LIN {X 0,Y 220.837,Z 392.973,A -85,B 0,C 180,E1 -20401.487,E2 -20401.487} C_VEL
LIN {X 0,Y 220.874,Z 392.97,A -85,B 0,C 180,E1 -20405.566,E2 -20405.566} C_VEL
LIN {X 0,Y 220.912,Z 392.963,A -85,B 0,C 180,E1 -20409.516,E2 -20409.516} C_VEL
LIN {X 0,Y 221.019,Z 392.952,A -85,B 0,C 180,E1 -20413.371,E2 -20413.371} C_VEL
LIN {X 0,Y 221.114,Z 392.939,A -85,B 0,C 180,E1 -20419.006,E2 -20419.006} C_VEL
LIN {X 0,Y 221.291,Z 392.918,A -85,B 0,C 180,E1 -20422.702,E2 -20422.702} C_VEL
LIN {X 0,Y 221.515,Z 392.893,A -85,B 0,C 180,E1 -20428.182,E2 -20428.182} C_VEL
LIN {X 0,Y 221.515,Z 392.893,A -85,B 0,C 180,E1 -20431.818,E2 -20431.818} C_VEL
LIN {X 0,Y 221.262,Z 392.922,A -85,B 0,C 180,E1 -20437.3,E2 -20437.3} C_VEL
LIN {X 0,Y 221.084,Z 392.943,A -85,B 0,C 180,E1 -20440.996,E2 -20440.996} C_VEL
LIN {X 0,Y 221.019,Z 392.952,A -85,B 0,C 180,E1 -20446.63,E2 -20446.63} C_VEL
LIN {X 0,Y 220.896,Z 392.965,A -85,B 0,C 180,E1 -20450.486,E2 -20450.486} C_VEL
LIN {X 0,Y 220.87,Z 392.97,A -85,B 0,C 180,E1 -20454.435,E2 -20454.435} C_VEL
LIN {X 0,Y 220.838,Z 392.973,A -85,B 0,C 180,E1 -20458.514,E2 -20458.514} C_VEL
LIN {X 0,Y 220.827,Z 392.976,A -85,B 0,C 180,E1 -20462.755,E2 -20462.755} C_VEL
LIN {X 0,Y 220.841,Z 392.976,A -85,B 0,C 180,E1 -20467.288,E2 -20467.288} C_VEL
LIN {X 0,Y 220.778,Z 392.982,A -85,B 0,C 180,E1 -20471.951,E2 -20471.951} C_VEL
LIN {X 0,Y 220.778,Z 392.982,A -85,B 0,C 180,E1 -20475.547,E2 -20475.547} C_VEL
LIN {X 0,Y 220.809,Z 392.978,A -85,B 0,C 180,E1 -20480.463,E2 -20480.463} C_VEL
LIN {X 0,Y 220.897,Z 392.967,A -85,B 0,C 180,E1 -20485.062,E2 -20485.062} C_VEL
LIN {X 0,Y 221.191,Z 393.123,A -85,B 0,C 180,E1 -20488.024,E2 -20488.024} C_VEL
LIN {X 0,Y 221.094,Z 396.042,A -85,B 0,C 180,E1 -20490.481,E2 -20490.481} C_VEL
LIN {X 0,Y 220.516,Z 400.977,A -85,B 0,C 180,E1 -20494.516,E2 -20494.516} C_VEL
LIN {X 0,Y 219.978,Z 407.083,A -85,B 0,C 180,E1 -20499.425,E2 -20499.425} C_VEL
LIN {X 0,Y 219.573,Z 412.628,A -85,B 0,C 180,E1 -20503.788,E2 -20503.788} C_VEL
LIN {X 0,Y 219.439,Z 417.082,A -85,B 0,C 180,E1 -20507.162,E2 -20507.162} C_VEL
LIN {X 0,Y 220.425,Z 428.94,A -85,B 0,C 180,E1 -20508.389,E2 -20508.389} C_VEL
LIN {X 0,Y 221.015,Z 435.556,A -85,B 0,C 180,E1 -20509.233,E2 -20509.233} C_VEL
LIN {X 0,Y 220.496,Z 447.027,A -85,B 0,C 180,E1 -20511.038,E2 -20511.038} C_VEL
LIN {X 0,Y 220.001,Z 457.347,A -85,B 0,C 180,E1 -20513.12,E2 -20513.12} C_VEL
LIN {X 0,Y 219.741,Z 464.712,A -85,B 0,C 180,E1 -20514.954,E2 -20514.954} C_VEL
LIN {X 0,Y 219.303,Z 472.284,A -85,B 0,C 180,E1 -20517.245,E2 -20517.245} C_VEL
LIN {X 0,Y 219.233,Z 478.476,A -85,B 0,C 180,E1 -20519.541,E2 -20519.541} C_VEL
LIN {X 0,Y 219.511,Z 483.38,A -85,B 0,C 180,E1 -20521.835,E2 -20521.835} C_VEL
LIN {X 0,Y 220.284,Z 487.936,A -85,B 0,C 180,E1 -20524.575,E2 -20524.575} C_VEL
LIN {X 0,Y 221.64,Z 491.134,A -85,B 0,C 180,E1 -20527.287,E2 -20527.287} C_VEL
LIN {X 0,Y 222.837,Z 492.539,A -85,B 0,C 180,E1 -20529.073,E2 -20529.073} C_VEL
LIN {X 0,Y 224.278,Z 493.429,A -85,B 0,C 180,E1 -20530.837,E2 -20530.837} C_VEL
LIN {X 0,Y 226.104,Z 493.732,A -85,B 0,C 180,E1 -20532.567,E2 -20532.567} C_VEL
LIN {X 0,Y 228.077,Z 493.509,A -85,B 0,C 180,E1 -20534.271,E2 -20534.271} C_VEL
LIN {X 0,Y 230.273,Z 492.801,A -85,B 0,C 180,E1 -20535.943,E2 -20535.943} C_VEL
LIN {X 0,Y 232.689,Z 491.534,A -85,B 0,C 180,E1 -20537.58,E2 -20537.58} C_VEL
LIN {X 0,Y 236.667,Z 488.649,A -85,B 0,C 180,E1 -20539.968,E2 -20539.968} C_VEL
LIN {X 0,Y 241.113,Z 484.562,A -85,B 0,C 180,E1 -20542.267,E2 -20542.267} C_VEL
LIN {X 0,Y 244.319,Z 481.041,A -85,B 0,C 180,E1 -20543.748,E2 -20543.748} C_VEL
LIN {X 0,Y 246.024,Z 477.848,A -85,B 0,C 180,E1 -20545.372,E2 -20545.372} C_VEL
LIN {X 0,Y 247.77,Z 472.241,A -85,B 0,C 180,E1 -20548.439,E2 -20548.439} C_VEL
LIN {X 0,Y 248.776,Z 467.147,A -85,B 0,C 180,E1 -20551.482,E2 -20551.482} C_VEL
LIN {X 0,Y 249.086,Z 464.573,A -85,B 0,C 180,E1 -20553.264,E2 -20553.264} C_VEL
LIN {X 0,Y 249.164,Z 462.654,A -85,B 0,C 180,E1 -20555.116,E2 -20555.116} C_VEL
LIN {X 0,Y 249.105,Z 460.856,A -85,B 0,C 180,E1 -20557.817,E2 -20557.817} C_VEL
LIN {X 0,Y 249.25,Z 460.084,A -85,B 0,C 180,E1 -20560.43,E2 -20560.43} C_VEL
LIN {X 0,Y 249.561,Z 460.468,A -85,B 0,C 180,E1 -20562.928,E2 -20562.928} C_VEL
LIN {X 0,Y 249.989,Z 461.962,A -85,B 0,C 180,E1 -20565.345,E2 -20565.345} C_VEL
LIN {X 0,Y 251.219,Z 465.936,A -85,B 0,C 180,E1 -20569.055,E2 -20569.055} C_VEL
LIN {X 0,Y 251.946,Z 468.627,A -85,B 0,C 180,E1 -20570.815,E2 -20570.815} C_VEL
LIN {X 0,Y 252.423,Z 471.374,A -85,B 0,C 180,E1 -20572.227,E2 -20572.227} C_VEL
LIN {X 0,Y 250.398,Z 479.099,A -85,B 0,C 180,E1 -20574.484,E2 -20574.484} C_VEL
LIN {X 0,Y 247.406,Z 487.692,A -85,B 0,C 180,E1 -20576.883,E2 -20576.883} C_VEL
LIN {X 0,Y 244.808,Z 493.219,A -85,B 0,C 180,E1 -20578.404,E2 -20578.404} C_VEL
LIN {X 0,Y 239.832,Z 501.02,A -85,B 0,C 180,E1 -20580.604,E2 -20580.604} C_VEL
LIN {X 0,Y 234.051,Z 508.808,A -85,B 0,C 180,E1 -20583.353,E2 -20583.353} C_VEL
LIN {X 0,Y 231.481,Z 511.607,A -85,B 0,C 180,E1 -20584.482,E2 -20584.482} C_VEL
LIN {X 0,Y 225.685,Z 515.698,A -85,B 0,C 180,E1 -20586.229,E2 -20586.229} C_VEL
LIN {X 0,Y 220.118,Z 519.017,A -85,B 0,C 180,E1 -20588.141,E2 -20588.141} C_VEL
LIN {X 0,Y 217.954,Z 520.611,A -85,B 0,C 180,E1 -20589.505,E2 -20589.505} C_VEL
LIN {X 0,Y 215.082,Z 523.55,A -85,B 0,C 180,E1 -20592.897,E2 -20592.897} C_VEL
LIN {X 0,Y 213.022,Z 525.29,A -85,B 0,C 180,E1 -20596.647,E2 -20596.647} C_VEL
LIN {X 0,Y 212.308,Z 525.696,A -85,B 0,C 180,E1 -20600.472,E2 -20600.472} C_VEL
LIN {X 0,Y 212.513,Z 524.63,A -85,B 0,C 180,E1 -20604.306,E2 -20604.306} C_VEL
LIN {X 0,Y 212.841,Z 523.547,A -85,B 0,C 180,E1 -20606.213,E2 -20606.213} C_VEL
LIN {X 0,Y 213.518,Z 521.058,A -85,B 0,C 180,E1 -20609.057,E2 -20609.057} C_VEL
LIN {X 0,Y 213.859,Z 517.355,A -85,B 0,C 180,E1 -20611.883,E2 -20611.883} C_VEL
LIN {X 0,Y 213.773,Z 512.137,A -85,B 0,C 180,E1 -20614.714,E2 -20614.714} C_VEL
LIN {X 0,Y 213.693,Z 506.567,A -85,B 0,C 180,E1 -20617.084,E2 -20617.084} C_VEL
LIN {X 0,Y 213.821,Z 498.336,A -85,B 0,C 180,E1 -20619.888,E2 -20619.888} C_VEL
LIN {X 0,Y 214.203,Z 488.282,A -85,B 0,C 180,E1 -20622.554,E2 -20622.554} C_VEL
LIN {X 0,Y 214.869,Z 478.168,A -85,B 0,C 180,E1 -20624.684,E2 -20624.684} C_VEL
LIN {X 0,Y 215.276,Z 471.414,A -85,B 0,C 180,E1 -20625.867,E2 -20625.867} C_VEL
LIN {X 0,Y 214.305,Z 459.661,A -85,B 0,C 180,E1 -20627.479,E2 -20627.479} C_VEL
LIN {X 0,Y 213.616,Z 447.834,A -85,B 0,C 180,E1 -20628.736,E2 -20628.736} C_VEL
LIN {X 0,Y 213.55,Z 435.845,A -85,B 0,C 180,E1 -20629.714,E2 -20629.714} C_VEL
LIN {X 0,Y 215.596,Z 424.642,A -85,B 0,C 180,E1 -20636.108,E2 -20636.108} C_VEL
LIN {X 0,Y 217.998,Z 415.833,A -85,B 0,C 180,E1 -20641.052,E2 -20641.052} C_VEL
LIN {X 0,Y 218.142,Z 414.232,A -85,B 0,C 180,E1 -20641.952,E2 -20641.952} C_VEL
LIN {X 0,Y 216.248,Z 405.804,A -85,B 0,C 180,E1 -20646.958,E2 -20646.958} C_VEL
LIN {X 0,Y 214.577,Z 397.868,A -85,B 0,C 180,E1 -20651.831,E2 -20651.831} C_VEL
LIN {X 0,Y 213.832,Z 393.846,A -85,B 0,C 180,E1 -20654.536,E2 -20654.536} C_VEL
LIN {X 0,Y 213.723,Z 393.86,A -85,B 0,C 180,E1 -20659.141,E2 -20659.141} C_VEL
LIN {X 0,Y 213.753,Z 393.858,A -85,B 0,C 180,E1 -20663.713,E2 -20663.713} C_VEL
LIN {X 0,Y 213.77,Z 393.857,A -85,B 0,C 180,E1 -20668.263,E2 -20668.263} C_VEL
LIN {X 0,Y 213.826,Z 393.847,A -85,B 0,C 180,E1 -20672.603,E2 -20672.603} C_VEL
LIN {X 0,Y 213.852,Z 393.844,A -85,B 0,C 180,E1 -20676.953,E2 -20676.953} C_VEL
LIN {X 0,Y 213.944,Z 393.829,A -85,B 0,C 180,E1 -20682.804,E2 -20682.804} C_VEL
LIN {X 0,Y 213.981,Z 393.829,A -85,B 0,C 180,E1 -20686.708,E2 -20686.708} C_VEL
LIN {X 0,Y 214.197,Z 393.799,A -85,B 0,C 180,E1 -20690.558,E2 -20690.558} C_VEL
LIN {X 0,Y 214.249,Z 393.793,A -85,B 0,C 180,E1 -20692.46,E2 -20692.46} C_VEL
LIN {X 0,Y 214.449,Z 393.769,A -85,B 0,C 180,E1 -20698.122,E2 -20698.122} C_VEL
LIN {X 0,Y 214.552,Z 393.756,A -85,B 0,C 180,E1 -20700,E2 -20700} C_VEL
LIN {X 0,Y 214.447,Z 393.771,A -85,B 0,C 180,E1 -20701.878,E2 -20701.878} C_VEL
LIN {X 0,Y 214.249,Z 393.794,A -85,B 0,C 180,E1 -20707.54,E2 -20707.54} C_VEL
LIN {X 0,Y 214.048,Z 393.823,A -85,B 0,C 180,E1 -20711.362,E2 -20711.362} C_VEL
LIN {X 0,Y 213.935,Z 393.836,A -85,B 0,C 180,E1 -20715.237,E2 -20715.237} C_VEL
LIN {X 0,Y 213.869,Z 393.844,A -85,B 0,C 180,E1 -20719.185,E2 -20719.185} C_VEL
LIN {X 0,Y 213.848,Z 393.847,A -85,B 0,C 180,E1 -20723.227,E2 -20723.227} C_VEL
LIN {X 0,Y 213.829,Z 393.848,A -85,B 0,C 180,E1 -20727.45,E2 -20727.45} C_VEL
LIN {X 0,Y 213.777,Z 393.854,A -85,B 0,C 180,E1 -20731.736,E2 -20731.736} C_VEL
LIN {X 0,Y 213.744,Z 393.857,A -85,B 0,C 180,E1 -20736.288,E2 -20736.288} C_VEL
LIN {X 0,Y 213.713,Z 393.862,A -85,B 0,C 180,E1 -20741.125,E2 -20741.125} C_VEL
LIN {X 0,Y 213.708,Z 393.86,A -85,B 0,C 180,E1 -20743.678,E2 -20743.678} C_VEL
LIN {X 0,Y 213.71,Z 393.864,A -85,B 0,C 180,E1 -20746.343,E2 -20746.343} C_VEL
LIN {X 0,Y 213.737,Z 393.856,A -85,B 0,C 180,E1 -20751.336,E2 -20751.336} C_VEL
LIN {X 0,Y 213.771,Z 393.856,A -85,B 0,C 180,E1 -20756.021,E2 -20756.021} C_VEL
LIN {X 0,Y 213.782,Z 393.853,A -85,B 0,C 180,E1 -20760.454,E2 -20760.454} C_VEL
LIN {X 0,Y 213.806,Z 393.852,A -85,B 0,C 180,E1 -20764.703,E2 -20764.703} C_VEL
LIN {X 0,Y 213.843,Z 393.844,A -85,B 0,C 180,E1 -20768.807,E2 -20768.807} C_VEL
LIN {X 0,Y 213.947,Z 393.834,A -85,B 0,C 180,E1 -20772.804,E2 -20772.804} C_VEL
LIN {X 0,Y 213.983,Z 393.826,A -85,B 0,C 180,E1 -20776.709,E2 -20776.709} C_VEL
LIN {X 0,Y 214.169,Z 393.807,A -85,B 0,C 180,E1 -20780.557,E2 -20780.557} C_VEL
LIN {X 0,Y 214.229,Z 393.799,A -85,B 0,C 180,E1 -20782.46,E2 -20782.46} C_VEL
LIN {X 0,Y 214.448,Z 393.773,A -85,B 0,C 180,E1 -20788.122,E2 -20788.122} C_VEL
LIN {X 0,Y 214.557,Z 393.761,A -85,B 0,C 180,E1 -20790,E2 -20790} C_VEL
LIN {X 0,Y 214.448,Z 393.773,A -85,B 0,C 180,E1 -20791.878,E2 -20791.878} C_VEL
LIN {X 0,Y 214.201,Z 393.802,A -85,B 0,C 180,E1 -20797.542,E2 -20797.542} C_VEL
LIN {X 0,Y 214.01,Z 393.825,A -85,B 0,C 180,E1 -20801.364,E2 -20801.364} C_VEL
LIN {X 0,Y 213.937,Z 393.834,A -85,B 0,C 180,E1 -20805.237,E2 -20805.237} C_VEL
LIN {X 0,Y 213.871,Z 393.843,A -85,B 0,C 180,E1 -20809.185,E2 -20809.185} C_VEL
LIN {X 0,Y 213.85,Z 393.844,A -85,B 0,C 180,E1 -20813.227,E2 -20813.227} C_VEL
LIN {X 0,Y 213.831,Z 393.85,A -85,B 0,C 180,E1 -20817.45,E2 -20817.45} C_VEL
LIN {X 0,Y 213.782,Z 393.855,A -85,B 0,C 180,E1 -20821.736,E2 -20821.736} C_VEL
LIN {X 0,Y 213.755,Z 393.856,A -85,B 0,C 180,E1 -20826.287,E2 -20826.287} C_VEL
LIN {X 0,Y 213.72,Z 393.862,A -85,B 0,C 180,E1 -20831.124,E2 -20831.124} C_VEL
LIN {X 0,Y 213.712,Z 393.863,A -85,B 0,C 180,E1 -20833.678,E2 -20833.678} C_VEL
LIN {X 0,Y 213.71,Z 393.86,A -85,B 0,C 180,E1 -20836.344,E2 -20836.344} C_VEL
LIN {X 0,Y 213.737,Z 393.862,A -85,B 0,C 180,E1 -20841.336,E2 -20841.336} C_VEL
LIN {X 0,Y 214.031,Z 393.818,A -85,B 0,C 180,E1 -20847.194,E2 -20847.194} C_VEL
LIN {X 0,Y 214.158,Z 393.995,A -85,B 0,C 180,E1 -20848.05,E2 -20848.05} C_VEL
LIN {X 0,Y 214.035,Z 396.832,A -85,B 0,C 180,E1 -20850.492,E2 -20850.492} C_VEL
LIN {X 0,Y 213.308,Z 403.024,A -85,B 0,C 180,E1 -20855.679,E2 -20855.679} C_VEL
LIN {X 0,Y 212.782,Z 409.154,A -85,B 0,C 180,E1 -20860.713,E2 -20860.713} C_VEL
LIN {X 0,Y 212.369,Z 415.285,A -85,B 0,C 180,E1 -20865.629,E2 -20865.629} C_VEL
LIN {X 0,Y 212.342,Z 417.279,A -85,B 0,C 180,E1 -20867.212,E2 -20867.212} C_VEL
LIN {X 0,Y 213.576,Z 431.068,A -85,B 0,C 180,E1 -20868.733,E2 -20868.733} C_VEL
LIN {X 0,Y 213.93,Z 435.64,A -85,B 0,C 180,E1 -20869.351,E2 -20869.351} C_VEL
LIN {X 0,Y 213.428,Z 446.255,A -85,B 0,C 180,E1 -20871.071,E2 -20871.071} C_VEL
LIN {X 0,Y 212.946,Z 456.398,A -85,B 0,C 180,E1 -20873.129,E2 -20873.129} C_VEL
LIN {X 0,Y 212.615,Z 464.917,A -85,B 0,C 180,E1 -20875.26,E2 -20875.26} C_VEL
LIN {X 0,Y 212.225,Z 472.594,A -85,B 0,C 180,E1 -20877.628,E2 -20877.628} C_VEL
LIN {X 0,Y 212.233,Z 479.859,A -85,B 0,C 180,E1 -20880.474,E2 -20880.474} C_VEL
LIN {X 0,Y 212.64,Z 484.667,A -85,B 0,C 180,E1 -20882.842,E2 -20882.842} C_VEL
LIN {X 0,Y 213.582,Z 489.1,A -85,B 0,C 180,E1 -20885.665,E2 -20885.665} C_VEL
LIN {X 0,Y 214.601,Z 491.312,A -85,B 0,C 180,E1 -20887.527,E2 -20887.527} C_VEL
LIN {X 0,Y 215.856,Z 492.951,A -85,B 0,C 180,E1 -20889.369,E2 -20889.369} C_VEL
LIN {X 0,Y 217.355,Z 494.052,A -85,B 0,C 180,E1 -20891.187,E2 -20891.187} C_VEL
LIN {X 0,Y 219.226,Z 494.623,A -85,B 0,C 180,E1 -20892.968,E2 -20892.968} C_VEL
LIN {X 0,Y 221.303,Z 494.639,A -85,B 0,C 180,E1 -20894.718,E2 -20894.718} C_VEL
LIN {X 0,Y 223.58,Z 494.155,A -85,B 0,C 180,E1 -20896.434,E2 -20896.434} C_VEL
LIN {X 0,Y 226.106,Z 493.159,A -85,B 0,C 180,E1 -20898.109,E2 -20898.109} C_VEL
LIN {X 0,Y 230.231,Z 490.713,A -85,B 0,C 180,E1 -20900.551,E2 -20900.551} C_VEL
LIN {X 0,Y 234.838,Z 487.053,A -85,B 0,C 180,E1 -20902.895,E2 -20902.895} C_VEL
LIN {X 0,Y 238.186,Z 483.92,A -85,B 0,C 180,E1 -20904.399,E2 -20904.399} C_VEL
LIN {X 0,Y 239.438,Z 482.364,A -85,B 0,C 180,E1 -20905.189,E2 -20905.189} C_VEL
LIN {X 0,Y 241.512,Z 478.123,A -85,B 0,C 180,E1 -20907.749,E2 -20907.749} C_VEL
LIN {X 0,Y 243.002,Z 473.908,A -85,B 0,C 180,E1 -20910.405,E2 -20910.405} C_VEL
LIN {X 0,Y 244.081,Z 470.048,A -85,B 0,C 180,E1 -20913.167,E2 -20913.167} C_VEL
LIN {X 0,Y 244.456,Z 468.089,A -85,B 0,C 180,E1 -20915.099,E2 -20915.099} C_VEL
LIN {X 0,Y 244.601,Z 466.776,A -85,B 0,C 180,E1 -20917.113,E2 -20917.113} C_VEL
LIN {X 0,Y 244.753,Z 465.998,A -85,B 0,C 180,E1 -20919.177,E2 -20919.177} C_VEL
LIN {X 0,Y 245.103,Z 465.903,A -85,B 0,C 180,E1 -20921.796,E2 -20921.796} C_VEL
LIN {X 0,Y 245.476,Z 466.939,A -85,B 0,C 180,E1 -20924.294,E2 -20924.294} C_VEL
LIN {X 0,Y 245.926,Z 468.963,A -85,B 0,C 180,E1 -20926.696,E2 -20926.696} C_VEL
LIN {X 0,Y 246.716,Z 471.544,A -85,B 0,C 180,E1 -20929.066,E2 -20929.066} C_VEL
LIN {X 0,Y 247.32,Z 475.087,A -85,B 0,C 180,E1 -20931.305,E2 -20931.305} C_VEL
LIN {X 0,Y 247.341,Z 475.694,A -85,B 0,C 180,E1 -20931.619,E2 -20931.619} C_VEL
LIN {X 0,Y 245.205,Z 482.097,A -85,B 0,C 180,E1 -20933.613,E2 -20933.613} C_VEL
LIN {X 0,Y 241.251,Z 491.306,A -85,B 0,C 180,E1 -20936.392,E2 -20936.392} C_VEL
LIN {X 0,Y 237.333,Z 497.714,A -85,B 0,C 180,E1 -20938.29,E2 -20938.29} C_VEL
LIN {X 0,Y 231.235,Z 505.657,A -85,B 0,C 180,E1 -20940.902,E2 -20940.902} C_VEL
LIN {X 0,Y 226.595,Z 511.194,A -85,B 0,C 180,E1 -20943.273,E2 -20943.273} C_VEL
LIN {X 0,Y 221.355,Z 517.034,A -85,B 0,C 180,E1 -20946.617,E2 -20946.617} C_VEL
LIN {X 0,Y 217.954,Z 520.611,A -85,B 0,C 180,E1 -20949.505,E2 -20949.505} C_VEL
LIN {X 0,Y 215.956,Z 522.049,A -85,B 0,C 180,E1 -20950.935,E2 -20950.935} C_VEL
LIN {X 0,Y 211.242,Z 523.676,A -85,B 0,C 180,E1 -20953.243,E2 -20953.243} C_VEL
LIN {X 0,Y 207.005,Z 524.439,A -85,B 0,C 180,E1 -20955.684,E2 -20955.684} C_VEL
LIN {X 0,Y 205.791,Z 524.586,A -85,B 0,C 180,E1 -20957.282,E2 -20957.282} C_VEL
LIN {X 0,Y 205.332,Z 524.55,A -85,B 0,C 180,E1 -20960.146,E2 -20960.146} C_VEL
LIN {X 0,Y 205.4,Z 523.786,A -85,B 0,C 180,E1 -20962.873,E2 -20962.873} C_VEL
LIN {X 0,Y 205.925,Z 521.948,A -85,B 0,C 180,E1 -20966.086,E2 -20966.086} C_VEL
LIN {X 0,Y 206.661,Z 519.266,A -85,B 0,C 180,E1 -20969.025,E2 -20969.025} C_VEL
LIN {X 0,Y 206.938,Z 516.786,A -85,B 0,C 180,E1 -20970.973,E2 -20970.973} C_VEL
LIN {X 0,Y 206.92,Z 511.789,A -85,B 0,C 180,E1 -20973.895,E2 -20973.895} C_VEL
LIN {X 0,Y 206.831,Z 506.392,A -85,B 0,C 180,E1 -20976.34,E2 -20976.34} C_VEL
LIN {X 0,Y 206.88,Z 498.083,A -85,B 0,C 180,E1 -20979.316,E2 -20979.316} C_VEL
LIN {X 0,Y 207.164,Z 489.529,A -85,B 0,C 180,E1 -20981.744,E2 -20981.744} C_VEL
LIN {X 0,Y 207.665,Z 479.929,A -85,B 0,C 180,E1 -20983.953,E2 -20983.953} C_VEL
LIN {X 0,Y 208.223,Z 470.769,A -85,B 0,C 180,E1 -20985.665,E2 -20985.665} C_VEL
LIN {X 0,Y 207.17,Z 458.539,A -85,B 0,C 180,E1 -20987.394,E2 -20987.394} C_VEL
LIN {X 0,Y 206.448,Z 445.761,A -85,B 0,C 180,E1 -20988.765,E2 -20988.765} C_VEL
LIN {X 0,Y 206.493,Z 435.575,A -85,B 0,C 180,E1 -20989.613,E2 -20989.613} C_VEL
LIN {X 0,Y 208.85,Z 423.145,A -85,B 0,C 180,E1 -20997.019,E2 -20997.019} C_VEL
LIN {X 0,Y 210.867,Z 416.142,A -85,B 0,C 180,E1 -21001.104,E2 -21001.104} C_VEL
LIN {X 0,Y 210.941,Z 414.257,A -85,B 0,C 180,E1 -21002.213,E2 -21002.213} C_VEL
LIN {X 0,Y 209.106,Z 406.113,A -85,B 0,C 180,E1 -21007.227,E2 -21007.227} C_VEL
LIN {X 0,Y 207.349,Z 397.654,A -85,B 0,C 180,E1 -21012.679,E2 -21012.679} C_VEL
LIN {X 0,Y 206.797,Z 394.722,A -85,B 0,C 180,E1 -21014.626,E2 -21014.626} C_VEL
LIN {X 0,Y 206.667,Z 394.74,A -85,B 0,C 180,E1 -21019.75,E2 -21019.75} C_VEL
LIN {X 0,Y 206.732,Z 394.729,A -85,B 0,C 180,E1 -21024.695,E2 -21024.695} C_VEL
LIN {X 0,Y 206.708,Z 394.735,A -85,B 0,C 180,E1 -21029.336,E2 -21029.336} C_VEL
LIN {X 0,Y 206.733,Z 394.731,A -85,B 0,C 180,E1 -21033.772,E2 -21033.772} C_VEL
LIN {X 0,Y 206.759,Z 394.731,A -85,B 0,C 180,E1 -21038.043,E2 -21038.043} C_VEL
LIN {X 0,Y 206.874,Z 394.711,A -85,B 0,C 180,E1 -21042.197,E2 -21042.197} C_VEL
LIN {X 0,Y 206.915,Z 394.71,A -85,B 0,C 180,E1 -21046.246,E2 -21046.246} C_VEL
LIN {X 0,Y 207.133,Z 394.68,A -85,B 0,C 180,E1 -21050.233,E2 -21050.233} C_VEL
LIN {X 0,Y 207.19,Z 394.673,A -85,B 0,C 180,E1 -21052.202,E2 -21052.202} C_VEL
LIN {X 0,Y 207.386,Z 394.649,A -85,B 0,C 180,E1 -21058.058,E2 -21058.058} C_VEL
LIN {X 0,Y 207.516,Z 394.632,A -85,B 0,C 180,E1 -21060,E2 -21060} C_VEL
LIN {X 0,Y 207.384,Z 394.651,A -85,B 0,C 180,E1 -21061.942,E2 -21061.942} C_VEL
LIN {X 0,Y 207.19,Z 394.672,A -85,B 0,C 180,E1 -21067.798,E2 -21067.798} C_VEL
LIN {X 0,Y 206.984,Z 394.702,A -85,B 0,C 180,E1 -21071.755,E2 -21071.755} C_VEL
LIN {X 0,Y 206.868,Z 394.713,A -85,B 0,C 180,E1 -21075.771,E2 -21075.771} C_VEL
LIN {X 0,Y 206.801,Z 394.723,A -85,B 0,C 180,E1 -21079.868,E2 -21079.868} C_VEL
LIN {X 0,Y 206.764,Z 394.726,A -85,B 0,C 180,E1 -21084.072,E2 -21084.072} C_VEL
LIN {X 0,Y 206.745,Z 394.73,A -85,B 0,C 180,E1 -21088.419,E2 -21088.419} C_VEL
LIN {X 0,Y 206.703,Z 394.736,A -85,B 0,C 180,E1 -21092.957,E2 -21092.957} C_VEL
LIN {X 0,Y 206.681,Z 394.738,A -85,B 0,C 180,E1 -21097.74,E2 -21097.74} C_VEL
LIN {X 0,Y 206.643,Z 394.741,A -85,B 0,C 180,E1 -21101.563,E2 -21101.563} C_VEL
LIN {X 0,Y 206.636,Z 394.743,A -85,B 0,C 180,E1 -21105.581,E2 -21105.581} C_VEL
LIN {X 0,Y 206.668,Z 394.738,A -85,B 0,C 180,E1 -21109.751,E2 -21109.751} C_VEL
LIN {X 0,Y 206.732,Z 394.735,A -85,B 0,C 180,E1 -21114.696,E2 -21114.696} C_VEL
LIN {X 0,Y 206.724,Z 394.729,A -85,B 0,C 180,E1 -21119.34,E2 -21119.34} C_VEL
LIN {X 0,Y 206.736,Z 394.732,A -85,B 0,C 180,E1 -21123.773,E2 -21123.773} C_VEL
LIN {X 0,Y 206.78,Z 394.725,A -85,B 0,C 180,E1 -21128.046,E2 -21128.046} C_VEL
LIN {X 0,Y 206.88,Z 394.716,A -85,B 0,C 180,E1 -21132.198,E2 -21132.198} C_VEL
LIN {X 0,Y 206.917,Z 394.708,A -85,B 0,C 180,E1 -21136.246,E2 -21136.246} C_VEL
LIN {X 0,Y 207.108,Z 394.688,A -85,B 0,C 180,E1 -21140.232,E2 -21140.232} C_VEL
LIN {X 0,Y 207.17,Z 394.68,A -85,B 0,C 180,E1 -21142.202,E2 -21142.202} C_VEL
LIN {X 0,Y 207.385,Z 394.652,A -85,B 0,C 180,E1 -21148.058,E2 -21148.058} C_VEL
LIN {X 0,Y 207.522,Z 394.637,A -85,B 0,C 180,E1 -21150,E2 -21150} C_VEL
LIN {X 0,Y 207.385,Z 394.652,A -85,B 0,C 180,E1 -21151.942,E2 -21151.942} C_VEL
LIN {X 0,Y 207.144,Z 394.683,A -85,B 0,C 180,E1 -21157.8,E2 -21157.8} C_VEL
LIN {X 0,Y 206.934,Z 394.707,A -85,B 0,C 180,E1 -21161.758,E2 -21161.758} C_VEL
LIN {X 0,Y 206.87,Z 394.717,A -85,B 0,C 180,E1 -21165.771,E2 -21165.771} C_VEL
LIN {X 0,Y 206.803,Z 394.723,A -85,B 0,C 180,E1 -21169.868,E2 -21169.868} C_VEL
LIN {X 0,Y 206.766,Z 394.728,A -85,B 0,C 180,E1 -21174.072,E2 -21174.072} C_VEL
LIN {X 0,Y 206.746,Z 394.728,A -85,B 0,C 180,E1 -21178.419,E2 -21178.419} C_VEL
LIN {X 0,Y 206.712,Z 394.735,A -85,B 0,C 180,E1 -21182.956,E2 -21182.956} C_VEL
LIN {X 0,Y 206.724,Z 394.736,A -85,B 0,C 180,E1 -21185.32,E2 -21185.32} C_VEL
LIN {X 0,Y 206.669,Z 394.738,A -85,B 0,C 180,E1 -21190.25,E2 -21190.25} C_VEL
LIN {X 0,Y 206.638,Z 394.743,A -85,B 0,C 180,E1 -21194.419,E2 -21194.419} C_VEL
LIN {X 0,Y 206.666,Z 394.74,A -85,B 0,C 180,E1 -21199.75,E2 -21199.75} C_VEL
LIN {X 0,Y 206.79,Z 394.724,A -85,B 0,C 180,E1 -21204.706,E2 -21204.706} C_VEL
LIN {X 0,Y 207.103,Z 394.779,A -85,B 0,C 180,E1 -21208.036,E2 -21208.036} C_VEL
LIN {X 0,Y 206.967,Z 397.585,A -85,B 0,C 180,E1 -21210.503,E2 -21210.503} C_VEL
LIN {X 0,Y 206.217,Z 403.809,A -85,B 0,C 180,E1 -21215.86,E2 -21215.86} C_VEL
LIN {X 0,Y 205.666,Z 409.986,A -85,B 0,C 180,E1 -21221.057,E2 -21221.057} C_VEL
LIN {X 0,Y 205.246,Z 416.182,A -85,B 0,C 180,E1 -21226.132,E2 -21226.132} C_VEL
LIN {X 0,Y 205.32,Z 417.92,A -85,B 0,C 180,E1 -21227.396,E2 -21227.396} C_VEL
LIN {X 0,Y 206.333,Z 429.717,A -85,B 0,C 180,E1 -21228.705,E2 -21228.705} C_VEL
LIN {X 0,Y 206.846,Z 435.455,A -85,B 0,C 180,E1 -21229.477,E2 -21229.477} C_VEL
LIN {X 0,Y 206.321,Z 446.59,A -85,B 0,C 180,E1 -21231.327,E2 -21231.327} C_VEL
LIN {X 0,Y 205.852,Z 457.552,A -85,B 0,C 180,E1 -21233.629,E2 -21233.629} C_VEL
LIN {X 0,Y 205.507,Z 465.035,A -85,B 0,C 180,E1 -21235.587,E2 -21235.587} C_VEL
LIN {X 0,Y 205.146,Z 472.735,A -85,B 0,C 180,E1 -21238.037,E2 -21238.037} C_VEL
LIN {X 0,Y 205.217,Z 480.166,A -85,B 0,C 180,E1 -21240.981,E2 -21240.981} C_VEL
LIN {X 0,Y 205.801,Z 485.903,A -85,B 0,C 180,E1 -21243.916,E2 -21243.916} C_VEL
LIN {X 0,Y 207.009,Z 490.203,A -85,B 0,C 180,E1 -21246.824,E2 -21246.824} C_VEL
LIN {X 0,Y 208.883,Z 493.26,A -85,B 0,C 180,E1 -21249.685,E2 -21249.685} C_VEL
LIN {X 0,Y 210.424,Z 494.58,A -85,B 0,C 180,E1 -21251.56,E2 -21251.56} C_VEL
LIN {X 0,Y 212.345,Z 495.383,A -85,B 0,C 180,E1 -21253.396,E2 -21253.396} C_VEL
LIN {X 0,Y 214.514,Z 495.672,A -85,B 0,C 180,E1 -21255.195,E2 -21255.195} C_VEL
LIN {X 0,Y 216.897,Z 495.42,A -85,B 0,C 180,E1 -21256.955,E2 -21256.955} C_VEL
LIN {X 0,Y 219.508,Z 494.704,A -85,B 0,C 180,E1 -21258.673,E2 -21258.673} C_VEL
LIN {X 0,Y 222.308,Z 493.472,A -85,B 0,C 180,E1 -21260.35,E2 -21260.35} C_VEL
LIN {X 0,Y 226.964,Z 490.656,A -85,B 0,C 180,E1 -21262.772,E2 -21262.772} C_VEL
LIN {X 0,Y 232.058,Z 486.671,A -85,B 0,C 180,E1 -21265.087,E2 -21265.087} C_VEL
LIN {X 0,Y 233.537,Z 485.182,A -85,B 0,C 180,E1 -21265.872,E2 -21265.872} C_VEL
LIN {X 0,Y 235.929,Z 481.413,A -85,B 0,C 180,E1 -21268.465,E2 -21268.465} C_VEL
LIN {X 0,Y 237.638,Z 477.935,A -85,B 0,C 180,E1 -21270.945,E2 -21270.945} C_VEL
LIN {X 0,Y 238.696,Z 475.387,A -85,B 0,C 180,E1 -21272.958,E2 -21272.958} C_VEL
LIN {X 0,Y 239.319,Z 473.662,A -85,B 0,C 180,E1 -21274.687,E2 -21274.687} C_VEL
LIN {X 0,Y 239.595,Z 472.711,A -85,B 0,C 180,E1 -21275.92,E2 -21275.92} C_VEL
LIN {X 0,Y 239.881,Z 471.721,A -85,B 0,C 180,E1 -21277.971,E2 -21277.971} C_VEL
LIN {X 0,Y 240.264,Z 471.255,A -85,B 0,C 180,E1 -21280.488,E2 -21280.488} C_VEL
LIN {X 0,Y 240.7,Z 471.781,A -85,B 0,C 180,E1 -21283.117,E2 -21283.117} C_VEL
LIN {X 0,Y 241.071,Z 473.374,A -85,B 0,C 180,E1 -21285.598,E2 -21285.598} C_VEL
LIN {X 0,Y 241.881,Z 476.899,A -85,B 0,C 180,E1 -21289.065,E2 -21289.065} C_VEL
LIN {X 0,Y 242.192,Z 479.631,A -85,B 0,C 180,E1 -21290.884,E2 -21290.884} C_VEL
LIN {X 0,Y 239.846,Z 485.293,A -85,B 0,C 180,E1 -21292.811,E2 -21292.811} C_VEL
LIN {X 0,Y 235.65,Z 493.429,A -85,B 0,C 180,E1 -21295.482,E2 -21295.482} C_VEL
LIN {X 0,Y 231.47,Z 499.46,A -85,B 0,C 180,E1 -21297.388,E2 -21297.388} C_VEL
LIN {X 0,Y 225.134,Z 506.741,A -85,B 0,C 180,E1 -21300.034,E2 -21300.034} C_VEL
LIN {X 0,Y 220.328,Z 511.895,A -85,B 0,C 180,E1 -21302.45,E2 -21302.45} C_VEL
LIN {X 0,Y 216.133,Z 516.053,A -85,B 0,C 180,E1 -21304.993,E2 -21304.993} C_VEL
LIN {X 0,Y 211.572,Z 520.272,A -85,B 0,C 180,E1 -21308.568,E2 -21308.568} C_VEL
LIN {X 0,Y 208.276,Z 523.058,A -85,B 0,C 180,E1 -21312.32,E2 -21312.32} C_VEL
LIN {X 0,Y 206.109,Z 524.476,A -85,B 0,C 180,E1 -21316.19,E2 -21316.19} C_VEL
LIN {X 0,Y 205.791,Z 524.586,A -85,B 0,C 180,E1 -21317.282,E2 -21317.282} C_VEL
LIN {X 0,Y 204.811,Z 524.584,A -85,B 0,C 180,E1 -21318.907,E2 -21318.907} C_VEL
LIN {X 0,Y 201.839,Z 523.559,A -85,B 0,C 180,E1 -21321.554,E2 -21321.554} C_VEL
LIN {X 0,Y 199.646,Z 522.068,A -85,B 0,C 180,E1 -21323.707,E2 -21323.707} C_VEL
LIN {X 0,Y 198.948,Z 520.749,A -85,B 0,C 180,E1 -21325.369,E2 -21325.369} C_VEL
LIN {X 0,Y 199.007,Z 520.317,A -85,B 0,C 180,E1 -21325.93,E2 -21325.93} C_VEL
LIN {X 0,Y 199.844,Z 517.371,A -85,B 0,C 180,E1 -21328.992,E2 -21328.992} C_VEL
LIN {X 0,Y 200.108,Z 514.669,A -85,B 0,C 180,E1 -21331.006,E2 -21331.006} C_VEL
LIN {X 0,Y 200.074,Z 509.378,A -85,B 0,C 180,E1 -21334.028,E2 -21334.028} C_VEL
LIN {X 0,Y 199.962,Z 503.648,A -85,B 0,C 180,E1 -21336.559,E2 -21336.559} C_VEL
LIN {X 0,Y 200.055,Z 495.013,A -85,B 0,C 180,E1 -21339.576,E2 -21339.576} C_VEL
LIN {X 0,Y 200.31,Z 485.712,A -85,B 0,C 180,E1 -21342.152,E2 -21342.152} C_VEL
LIN {X 0,Y 200.937,Z 475.454,A -85,B 0,C 180,E1 -21344.43,E2 -21344.43} C_VEL
LIN {X 0,Y 201.179,Z 469.934,A -85,B 0,C 180,E1 -21345.448,E2 -21345.448} C_VEL
LIN {X 0,Y 200.083,Z 457.782,A -85,B 0,C 180,E1 -21347.224,E2 -21347.224} C_VEL
LIN {X 0,Y 199.39,Z 445.132,A -85,B 0,C 180,E1 -21348.628,E2 -21348.628} C_VEL
LIN {X 0,Y 199.414,Z 435.241,A -85,B 0,C 180,E1 -21349.494,E2 -21349.494} C_VEL
LIN {X 0,Y 201.679,Z 423.313,A -85,B 0,C 180,E1 -21356.937,E2 -21356.937} C_VEL
LIN {X 0,Y 203.715,Z 416.397,A -85,B 0,C 180,E1 -21361.164,E2 -21361.164} C_VEL
LIN {X 0,Y 203.57,Z 413.533,A -85,B 0,C 180,E1 -21362.939,E2 -21362.939} C_VEL
LIN {X 0,Y 201.814,Z 405.948,A -85,B 0,C 180,E1 -21367.812,E2 -21367.812} C_VEL
LIN {X 0,Y 200.362,Z 398.858,A -85,B 0,C 180,E1 -21372.557,E2 -21372.557} C_VEL
LIN {X 0,Y 199.72,Z 395.603,A -85,B 0,C 180,E1 -21374.89,E2 -21374.89} C_VEL
LIN {X 0,Y 199.641,Z 395.616,A -85,B 0,C 180,E1 -21380.756,E2 -21380.756} C_VEL
LIN {X 0,Y 199.634,Z 395.614,A -85,B 0,C 180,E1 -21385.718,E2 -21385.718} C_VEL
LIN {X 0,Y 199.697,Z 395.611,A -85,B 0,C 180,E1 -21388.136,E2 -21388.136} C_VEL
LIN {X 0,Y 199.686,Z 395.608,A -85,B 0,C 180,E1 -21392.772,E2 -21392.772} C_VEL
LIN {X 0,Y 199.739,Z 395.603,A -85,B 0,C 180,E1 -21397.229,E2 -21397.229} C_VEL
LIN {X 0,Y 199.797,Z 395.595,A -85,B 0,C 180,E1 -21401.757,E2 -21401.757} C_VEL
LIN {X 0,Y 199.849,Z 395.592,A -85,B 0,C 180,E1 -21405.749,E2 -21405.749} C_VEL
LIN {X 0,Y 200.076,Z 395.56,A -85,B 0,C 180,E1 -21409.884,E2 -21409.884} C_VEL
LIN {X 0,Y 200.133,Z 395.553,A -85,B 0,C 180,E1 -21411.925,E2 -21411.925} C_VEL
LIN {X 0,Y 200.325,Z 395.529,A -85,B 0,C 180,E1 -21417.99,E2 -21417.99} C_VEL
LIN {X 0,Y 200.481,Z 395.508,A -85,B 0,C 180,E1 -21420,E2 -21420} C_VEL
LIN {X 0,Y 200.033,Z 395.567,A -85,B 0,C 180,E1 -21424.029,E2 -21424.029} C_VEL
LIN {X 0,Y 200.133,Z 395.55,A -85,B 0,C 180,E1 -21428.075,E2 -21428.075} C_VEL
LIN {X 0,Y 199.916,Z 395.581,A -85,B 0,C 180,E1 -21432.177,E2 -21432.177} C_VEL
LIN {X 0,Y 199.807,Z 395.592,A -85,B 0,C 180,E1 -21436.343,E2 -21436.343} C_VEL
LIN {X 0,Y 199.824,Z 395.59,A -85,B 0,C 180,E1 -21438.454,E2 -21438.454} C_VEL
LIN {X 0,Y 199.737,Z 395.602,A -85,B 0,C 180,E1 -21443.817,E2 -21443.817} C_VEL
LIN {X 0,Y 199.713,Z 395.606,A -85,B 0,C 180,E1 -21448.387,E2 -21448.387} C_VEL
LIN {X 0,Y 199.678,Z 395.61,A -85,B 0,C 180,E1 -21452.359,E2 -21452.359} C_VEL
LIN {X 0,Y 199.623,Z 395.618,A -85,B 0,C 180,E1 -21456.763,E2 -21456.763} C_VEL
LIN {X 0,Y 199.609,Z 395.62,A -85,B 0,C 180,E1 -21459.328,E2 -21459.328} C_VEL
LIN {X 0,Y 199.575,Z 395.622,A -85,B 0,C 180,E1 -21462.311,E2 -21462.311} C_VEL
LIN {X 0,Y 199.583,Z 395.623,A -85,B 0,C 180,E1 -21465.23,E2 -21465.23} C_VEL
LIN {X 0,Y 199.64,Z 395.614,A -85,B 0,C 180,E1 -21470.68,E2 -21470.68} C_VEL
LIN {X 0,Y 199.636,Z 395.616,A -85,B 0,C 180,E1 -21475.718,E2 -21475.718} C_VEL
LIN {X 0,Y 199.705,Z 395.608,A -85,B 0,C 180,E1 -21478.138,E2 -21478.138} C_VEL
LIN {X 0,Y 199.689,Z 395.611,A -85,B 0,C 180,E1 -21482.772,E2 -21482.772} C_VEL
LIN {X 0,Y 199.752,Z 395.599,A -85,B 0,C 180,E1 -21487.231,E2 -21487.231} C_VEL
LIN {X 0,Y 199.839,Z 395.591,A -85,B 0,C 180,E1 -21491.722,E2 -21491.722} C_VEL
LIN {X 0,Y 199.851,Z 395.589,A -85,B 0,C 180,E1 -21495.75,E2 -21495.75} C_VEL
LIN {X 0,Y 200.072,Z 395.562,A -85,B 0,C 180,E1 -21499.885,E2 -21499.885} C_VEL
LIN {X 0,Y 200.036,Z 395.567,A -85,B 0,C 180,E1 -21503.95,E2 -21503.95} C_VEL
LIN {X 0,Y 200.324,Z 395.531,A -85,B 0,C 180,E1 -21507.99,E2 -21507.99} C_VEL
LIN {X 0,Y 200.486,Z 395.513,A -85,B 0,C 180,E1 -21510,E2 -21510} C_VEL
LIN {X 0,Y 200.031,Z 395.565,A -85,B 0,C 180,E1 -21514.03,E2 -21514.03} C_VEL
LIN {X 0,Y 200.092,Z 395.561,A -85,B 0,C 180,E1 -21518.077,E2 -21518.077} C_VEL
LIN {X 0,Y 199.882,Z 395.582,A -85,B 0,C 180,E1 -21522.179,E2 -21522.179} C_VEL
LIN {X 0,Y 199.809,Z 395.595,A -85,B 0,C 180,E1 -21526.344,E2 -21526.344} C_VEL
LIN {X 0,Y 199.826,Z 395.592,A -85,B 0,C 180,E1 -21528.454,E2 -21528.454} C_VEL
LIN {X 0,Y 199.74,Z 395.605,A -85,B 0,C 180,E1 -21533.818,E2 -21533.818} C_VEL
LIN {X 0,Y 199.715,Z 395.604,A -85,B 0,C 180,E1 -21538.387,E2 -21538.387} C_VEL
LIN {X 0,Y 199.667,Z 395.611,A -85,B 0,C 180,E1 -21542.353,E2 -21542.353} C_VEL
LIN {X 0,Y 199.642,Z 395.614,A -85,B 0,C 180,E1 -21546.76,E2 -21546.76} C_VEL
LIN {X 0,Y 199.641,Z 395.614,A -85,B 0,C 180,E1 -21549.321,E2 -21549.321} C_VEL
LIN {X 0,Y 199.584,Z 395.623,A -85,B 0,C 180,E1 -21554.771,E2 -21554.771} C_VEL
LIN {X 0,Y 199.583,Z 395.62,A -85,B 0,C 180,E1 -21558.005,E2 -21558.005} C_VEL
LIN {X 0,Y 199.643,Z 395.616,A -85,B 0,C 180,E1 -21560.757,E2 -21560.757} C_VEL
LIN {X 0,Y 199.813,Z 395.589,A -85,B 0,C 180,E1 -21565.753,E2 -21565.753} C_VEL
LIN {X 0,Y 200.058,Z 395.76,A -85,B 0,C 180,E1 -21568.2,E2 -21568.2} C_VEL
LIN {X 0,Y 199.726,Z 399.535,A -85,B 0,C 180,E1 -21571.608,E2 -21571.608} C_VEL
LIN {X 0,Y 198.981,Z 405.818,A -85,B 0,C 180,E1 -21577.138,E2 -21577.138} C_VEL
LIN {X 0,Y 198.536,Z 410.795,A -85,B 0,C 180,E1 -21581.422,E2 -21581.422} C_VEL
LIN {X 0,Y 198.229,Z 418.045,A -85,B 0,C 180,E1 -21587.523,E2 -21587.523} C_VEL
LIN {X 0,Y 199.316,Z 430.422,A -85,B 0,C 180,E1 -21588.946,E2 -21588.946} C_VEL
LIN {X 0,Y 199.768,Z 435.24,A -85,B 0,C 180,E1 -21589.613,E2 -21589.613} C_VEL
LIN {X 0,Y 199.23,Z 446.944,A -85,B 0,C 180,E1 -21591.62,E2 -21591.62} C_VEL
LIN {X 0,Y 198.828,Z 457.422,A -85,B 0,C 180,E1 -21593.913,E2 -21593.913} C_VEL
LIN {X 0,Y 198.362,Z 466.688,A -85,B 0,C 180,E1 -21596.445,E2 -21596.445} C_VEL
LIN {X 0,Y 198.102,Z 475.581,A -85,B 0,C 180,E1 -21599.492,E2 -21599.492} C_VEL
LIN {X 0,Y 198.391,Z 482.464,A -85,B 0,C 180,E1 -21602.538,E2 -21602.538} C_VEL
LIN {X 0,Y 199.07,Z 487.064,A -85,B 0,C 180,E1 -21605.064,E2 -21605.064} C_VEL
LIN {X 0,Y 200.528,Z 491.293,A -85,B 0,C 180,E1 -21608.059,E2 -21608.059} C_VEL
LIN {X 0,Y 201.9,Z 493.401,A -85,B 0,C 180,E1 -21610.023,E2 -21610.023} C_VEL
LIN {X 0,Y 203.491,Z 495,A -85,B 0,C 180,E1 -21611.96,E2 -21611.96} C_VEL
LIN {X 0,Y 205.467,Z 496.039,A -85,B 0,C 180,E1 -21613.853,E2 -21613.853} C_VEL
LIN {X 0,Y 207.737,Z 496.574,A -85,B 0,C 180,E1 -21615.703,E2 -21615.703} C_VEL
LIN {X 0,Y 210.204,Z 496.599,A -85,B 0,C 180,E1 -21617.512,E2 -21617.512} C_VEL
LIN {X 0,Y 212.903,Z 496.118,A -85,B 0,C 180,E1 -21619.275,E2 -21619.275} C_VEL
LIN {X 0,Y 215.828,Z 495.178,A -85,B 0,C 180,E1 -21620.989,E2 -21620.989} C_VEL
LIN {X 0,Y 219,Z 493.715,A -85,B 0,C 180,E1 -21622.65,E2 -21622.65} C_VEL
LIN {X 0,Y 224.135,Z 490.584,A -85,B 0,C 180,E1 -21625.044,E2 -21625.044} C_VEL
LIN {X 0,Y 227.611,Z 487.945,A -85,B 0,C 180,E1 -21626.598,E2 -21626.598} C_VEL
LIN {X 0,Y 229.501,Z 485.702,A -85,B 0,C 180,E1 -21628.337,E2 -21628.337} C_VEL
LIN {X 0,Y 231.783,Z 482.377,A -85,B 0,C 180,E1 -21631.029,E2 -21631.029} C_VEL
LIN {X 0,Y 233.061,Z 480.232,A -85,B 0,C 180,E1 -21632.874,E2 -21632.874} C_VEL
LIN {X 0,Y 234.018,Z 478.456,A -85,B 0,C 180,E1 -21634.793,E2 -21634.793} C_VEL
LIN {X 0,Y 234.594,Z 477.272,A -85,B 0,C 180,E1 -21636.81,E2 -21636.81} C_VEL
LIN {X 0,Y 235.017,Z 476.584,A -85,B 0,C 180,E1 -21638.966,E2 -21638.966} C_VEL
LIN {X 0,Y 235.603,Z 476.584,A -85,B 0,C 180,E1 -21641.776,E2 -21641.776} C_VEL
LIN {X 0,Y 236.004,Z 477.666,A -85,B 0,C 180,E1 -21644.381,E2 -21644.381} C_VEL
LIN {X 0,Y 236.52,Z 480.787,A -85,B 0,C 180,E1 -21647.975,E2 -21647.975} C_VEL
LIN {X 0,Y 236.824,Z 483.205,A -85,B 0,C 180,E1 -21649.967,E2 -21649.967} C_VEL
LIN {X 0,Y 236.44,Z 484.549,A -85,B 0,C 180,E1 -21650.609,E2 -21650.609} C_VEL
LIN {X 0,Y 232.96,Z 490.882,A -85,B 0,C 180,E1 -21652.888,E2 -21652.888} C_VEL
LIN {X 0,Y 229.268,Z 496.629,A -85,B 0,C 180,E1 -21654.916,E2 -21654.916} C_VEL
LIN {X 0,Y 223.709,Z 503.109,A -85,B 0,C 180,E1 -21657.185,E2 -21657.185} C_VEL
LIN {X 0,Y 217.304,Z 509.509,A -85,B 0,C 180,E1 -21659.914,E2 -21659.914} C_VEL
LIN {X 0,Y 211.159,Z 515.142,A -85,B 0,C 180,E1 -21663.299,E2 -21663.299} C_VEL
LIN {X 0,Y 207.179,Z 518.38,A -85,B 0,C 180,E1 -21665.979,E2 -21665.979} C_VEL
LIN {X 0,Y 203.104,Z 521.466,A -85,B 0,C 180,E1 -21669.755,E2 -21669.755} C_VEL
LIN {X 0,Y 200.257,Z 523.197,A -85,B 0,C 180,E1 -21673.694,E2 -21673.694} C_VEL
LIN {X 0,Y 198.661,Z 523.619,A -85,B 0,C 180,E1 -21677.745,E2 -21677.745} C_VEL
LIN {X 0,Y 198.388,Z 522.675,A -85,B 0,C 180,E1 -21681.853,E2 -21681.853} C_VEL
LIN {X 0,Y 198.599,Z 521.699,A -85,B 0,C 180,E1 -21683.905,E2 -21683.905} C_VEL
LIN {X 0,Y 199.007,Z 520.317,A -85,B 0,C 180,E1 -21685.93,E2 -21685.93} C_VEL
LIN {X 0,Y 198.968,Z 519.36,A -85,B 0,C 180,E1 -21687.028,E2 -21687.028} C_VEL
LIN {X 0,Y 197.982,Z 517.345,A -85,B 0,C 180,E1 -21688.612,E2 -21688.612} C_VEL
LIN {X 0,Y 196.404,Z 514.852,A -85,B 0,C 180,E1 -21690.124,E2 -21690.124} C_VEL
LIN {X 0,Y 194.244,Z 510.982,A -85,B 0,C 180,E1 -21692.13,E2 -21692.13} C_VEL
LIN {X 0,Y 193.337,Z 507.863,A -85,B 0,C 180,E1 -21693.651,E2 -21693.651} C_VEL
LIN {X 0,Y 193.285,Z 506.783,A -85,B 0,C 180,E1 -21694.164,E2 -21694.164} C_VEL
LIN {X 0,Y 193.087,Z 500.632,A -85,B 0,C 180,E1 -21696.793,E2 -21696.793} C_VEL
LIN {X 0,Y 193.176,Z 492.785,A -85,B 0,C 180,E1 -21699.532,E2 -21699.532} C_VEL
LIN {X 0,Y 193.413,Z 483.934,A -85,B 0,C 180,E1 -21702.006,E2 -21702.006} C_VEL
LIN {X 0,Y 194.062,Z 473.19,A -85,B 0,C 180,E1 -21704.417,E2 -21704.417} C_VEL
LIN {X 0,Y 194.141,Z 468.9,A -85,B 0,C 180,E1 -21705.215,E2 -21705.215} C_VEL
LIN {X 0,Y 193.053,Z 457.577,A -85,B 0,C 180,E1 -21706.932,E2 -21706.932} C_VEL
LIN {X 0,Y 192.339,Z 444.586,A -85,B 0,C 180,E1 -21708.442,E2 -21708.442} C_VEL
LIN {X 0,Y 192.345,Z 434.967,A -85,B 0,C 180,E1 -21709.337,E2 -21709.337} C_VEL
LIN {X 0,Y 194.516,Z 423.463,A -85,B 0,C 180,E1 -21716.848,E2 -21716.848} C_VEL
LIN {X 0,Y 196.634,Z 416.251,A -85,B 0,C 180,E1 -21721.463,E2 -21721.463} C_VEL
LIN {X 0,Y 196.651,Z 414.758,A -85,B 0,C 180,E1 -21722.417,E2 -21722.417} C_VEL
LIN {X 0,Y 194.865,Z 407.155,A -85,B 0,C 180,E1 -21727.491,E2 -21727.491} C_VEL
LIN {X 0,Y 193.156,Z 398.772,A -85,B 0,C 180,E1 -21733.306,E2 -21733.306} C_VEL
LIN {X 0,Y 192.675,Z 396.48,A -85,B 0,C 180,E1 -21735.061,E2 -21735.061} C_VEL
LIN {X 0,Y 192.543,Z 396.501,A -85,B 0,C 180,E1 -21740.042,E2 -21740.042} C_VEL
LIN {X 0,Y 192.598,Z 396.491,A -85,B 0,C 180,E1 -21744.278,E2 -21744.278} C_VEL
LIN {X 0,Y 192.6,Z 396.492,A -85,B 0,C 180,E1 -21749.279,E2 -21749.279} C_VEL
LIN {X 0,Y 192.661,Z 396.486,A -85,B 0,C 180,E1 -21751.691,E2 -21751.691} C_VEL
LIN {X 0,Y 192.706,Z 396.479,A -85,B 0,C 180,E1 -21756.349,E2 -21756.349} C_VEL
LIN {X 0,Y 192.732,Z 396.476,A -85,B 0,C 180,E1 -21761.457,E2 -21761.457} C_VEL
LIN {X 0,Y 192.773,Z 396.47,A -85,B 0,C 180,E1 -21765.214,E2 -21765.214} C_VEL
LIN {X 0,Y 193.021,Z 396.441,A -85,B 0,C 180,E1 -21769.511,E2 -21769.511} C_VEL
LIN {X 0,Y 193.006,Z 396.444,A -85,B 0,C 180,E1 -21773.729,E2 -21773.729} C_VEL
LIN {X 0,Y 193.267,Z 396.408,A -85,B 0,C 180,E1 -21777.916,E2 -21777.916} C_VEL
LIN {X 0,Y 193.445,Z 396.384,A -85,B 0,C 180,E1 -21780,E2 -21780} C_VEL
LIN {X 0,Y 192.98,Z 396.445,A -85,B 0,C 180,E1 -21784.177,E2 -21784.177} C_VEL
LIN {X 0,Y 193.08,Z 396.428,A -85,B 0,C 180,E1 -21788.372,E2 -21788.372} C_VEL
LIN {X 0,Y 192.854,Z 396.461,A -85,B 0,C 180,E1 -21792.63,E2 -21792.63} C_VEL
LIN {X 0,Y 192.782,Z 396.467,A -85,B 0,C 180,E1 -21798.586,E2 -21798.586} C_VEL
LIN {X 0,Y 192.665,Z 396.482,A -85,B 0,C 180,E1 -21804.225,E2 -21804.225} C_VEL
LIN {X 0,Y 192.65,Z 396.488,A -85,B 0,C 180,E1 -21808.892,E2 -21808.892} C_VEL
LIN {X 0,Y 192.599,Z 396.49,A -85,B 0,C 180,E1 -21813.186,E2 -21813.186} C_VEL
LIN {X 0,Y 192.552,Z 396.499,A -85,B 0,C 180,E1 -21818.352,E2 -21818.352} C_VEL
LIN {X 0,Y 192.493,Z 396.504,A -85,B 0,C 180,E1 -21823.096,E2 -21823.096} C_VEL
LIN {X 0,Y 192.515,Z 396.505,A -85,B 0,C 180,E1 -21826.897,E2 -21826.897} C_VEL
LIN {X 0,Y 192.575,Z 396.491,A -85,B 0,C 180,E1 -21831.654,E2 -21831.654} C_VEL
LIN {X 0,Y 192.599,Z 396.493,A -85,B 0,C 180,E1 -21834.279,E2 -21834.279} C_VEL
LIN {X 0,Y 192.609,Z 396.488,A -85,B 0,C 180,E1 -21839.281,E2 -21839.281} C_VEL
LIN {X 0,Y 192.666,Z 396.482,A -85,B 0,C 180,E1 -21841.692,E2 -21841.692} C_VEL
LIN {X 0,Y 192.713,Z 396.48,A -85,B 0,C 180,E1 -21846.35,E2 -21846.35} C_VEL
LIN {X 0,Y 192.783,Z 396.469,A -85,B 0,C 180,E1 -21851.414,E2 -21851.414} C_VEL
LIN {X 0,Y 192.855,Z 396.456,A -85,B 0,C 180,E1 -21857.371,E2 -21857.371} C_VEL
LIN {X 0,Y 193.064,Z 396.435,A -85,B 0,C 180,E1 -21861.628,E2 -21861.628} C_VEL
LIN {X 0,Y 193.266,Z 396.41,A -85,B 0,C 180,E1 -21867.916,E2 -21867.916} C_VEL
LIN {X 0,Y 193.449,Z 396.39,A -85,B 0,C 180,E1 -21870,E2 -21870} C_VEL
LIN {X 0,Y 192.977,Z 396.443,A -85,B 0,C 180,E1 -21874.177,E2 -21874.177} C_VEL
LIN {X 0,Y 193.039,Z 396.439,A -85,B 0,C 180,E1 -21878.374,E2 -21878.374} C_VEL
LIN {X 0,Y 192.808,Z 396.462,A -85,B 0,C 180,E1 -21882.633,E2 -21882.633} C_VEL
LIN {X 0,Y 192.774,Z 396.471,A -85,B 0,C 180,E1 -21886.958,E2 -21886.958} C_VEL
LIN {X 0,Y 192.646,Z 396.485,A -85,B 0,C 180,E1 -21891.397,E2 -21891.397} C_VEL
LIN {X 0,Y 192.667,Z 396.484,A -85,B 0,C 180,E1 -21894.225,E2 -21894.225} C_VEL
LIN {X 0,Y 192.652,Z 396.484,A -85,B 0,C 180,E1 -21898.892,E2 -21898.892} C_VEL
LIN {X 0,Y 192.603,Z 396.493,A -85,B 0,C 180,E1 -21903.186,E2 -21903.186} C_VEL
LIN {X 0,Y 192.612,Z 396.49,A -85,B 0,C 180,E1 -21906.608,E2 -21906.608} C_VEL
LIN {X 0,Y 192.527,Z 396.502,A -85,B 0,C 180,E1 -21911.078,E2 -21911.078} C_VEL
LIN {X 0,Y 192.495,Z 396.502,A -85,B 0,C 180,E1 -21916.077,E2 -21916.077} C_VEL
LIN {X 0,Y 192.542,Z 396.499,A -85,B 0,C 180,E1 -21920.043,E2 -21920.043} C_VEL
LIN {X 0,Y 192.654,Z 396.484,A -85,B 0,C 180,E1 -21924.29,E2 -21924.29} C_VEL
LIN {X 0,Y 193.009,Z 396.604,A -85,B 0,C 180,E1 -21928.284,E2 -21928.284} C_VEL
LIN {X 0,Y 192.614,Z 400.288,A -85,B 0,C 180,E1 -21931.684,E2 -21931.684} C_VEL
LIN {X 0,Y 191.861,Z 406.57,A -85,B 0,C 180,E1 -21937.38,E2 -21937.38} C_VEL
LIN {X 0,Y 191.289,Z 412.688,A -85,B 0,C 180,E1 -21942.796,E2 -21942.796} C_VEL
LIN {X 0,Y 191.197,Z 418.474,A -85,B 0,C 180,E1 -21947.731,E2 -21947.731} C_VEL
LIN {X 0,Y 192.292,Z 430.779,A -85,B 0,C 180,E1 -21949.204,E2 -21949.204} C_VEL
LIN {X 0,Y 192.652,Z 436.585,A -85,B 0,C 180,E1 -21950.055,E2 -21950.055} C_VEL
LIN {X 0,Y 192.122,Z 447.91,A -85,B 0,C 180,E1 -21952.115,E2 -21952.115} C_VEL
LIN {X 0,Y 191.745,Z 458.279,A -85,B 0,C 180,E1 -21954.479,E2 -21954.479} C_VEL
LIN {X 0,Y 191.282,Z 466.655,A -85,B 0,C 180,E1 -21956.841,E2 -21956.841} C_VEL
LIN {X 0,Y 191.085,Z 474.227,A -85,B 0,C 180,E1 -21959.473,E2 -21959.473} C_VEL
LIN {X 0,Y 191.358,Z 481.588,A -85,B 0,C 180,E1 -21962.631,E2 -21962.631} C_VEL
LIN {X 0,Y 192.015,Z 486.486,A -85,B 0,C 180,E1 -21965.25,E2 -21965.25} C_VEL
LIN {X 0,Y 193.499,Z 491.08,A -85,B 0,C 180,E1 -21968.354,E2 -21968.354} C_VEL
LIN {X 0,Y 194.91,Z 493.432,A -85,B 0,C 180,E1 -21970.387,E2 -21970.387} C_VEL
LIN {X 0,Y 196.572,Z 495.271,A -85,B 0,C 180,E1 -21972.387,E2 -21972.387} C_VEL
LIN {X 0,Y 198.602,Z 496.57,A -85,B 0,C 180,E1 -21974.342,E2 -21974.342} C_VEL
LIN {X 0,Y 200.94,Z 497.348,A -85,B 0,C 180,E1 -21976.249,E2 -21976.249} C_VEL
LIN {X 0,Y 203.504,Z 497.651,A -85,B 0,C 180,E1 -21978.108,E2 -21978.108} C_VEL
LIN {X 0,Y 206.31,Z 497.432,A -85,B 0,C 180,E1 -21979.917,E2 -21979.917} C_VEL
LIN {X 0,Y 209.359,Z 496.767,A -85,B 0,C 180,E1 -21981.67,E2 -21981.67} C_VEL
LIN {X 0,Y 212.646,Z 495.581,A -85,B 0,C 180,E1 -21983.366,E2 -21983.366} C_VEL
LIN {X 0,Y 217.978,Z 492.936,A -85,B 0,C 180,E1 -21985.802,E2 -21985.802} C_VEL
LIN {X 0,Y 222.032,Z 490.295,A -85,B 0,C 180,E1 -21987.589,E2 -21987.589} C_VEL
LIN {X 0,Y 224.666,Z 487.633,A -85,B 0,C 180,E1 -21990.034,E2 -21990.034} C_VEL
LIN {X 0,Y 226.304,Z 485.689,A -85,B 0,C 180,E1 -21991.867,E2 -21991.867} C_VEL
LIN {X 0,Y 227.748,Z 483.929,A -85,B 0,C 180,E1 -21993.742,E2 -21993.742} C_VEL
LIN {X 0,Y 228.816,Z 482.482,A -85,B 0,C 180,E1 -21995.703,E2 -21995.703} C_VEL
LIN {X 0,Y 229.409,Z 481.651,A -85,B 0,C 180,E1 -21997.786,E2 -21997.786} C_VEL
LIN {X 0,Y 230.038,Z 481.328,A -85,B 0,C 180,E1 -22000.2,E2 -22000.2} C_VEL
LIN {X 0,Y 230.638,Z 481.84,A -85,B 0,C 180,E1 -22003.002,E2 -22003.002} C_VEL
LIN {X 0,Y 230.89,Z 483.419,A -85,B 0,C 180,E1 -22005.565,E2 -22005.565} C_VEL
LIN {X 0,Y 231.178,Z 485.631,A -85,B 0,C 180,E1 -22008.024,E2 -22008.024} C_VEL
LIN {X 0,Y 231.294,Z 487.191,A -85,B 0,C 180,E1 -22009.433,E2 -22009.433} C_VEL
LIN {X 0,Y 230.042,Z 489.539,A -85,B 0,C 180,E1 -22010.463,E2 -22010.463} C_VEL
LIN {X 0,Y 225.351,Z 496.338,A -85,B 0,C 180,E1 -22013.105,E2 -22013.105} C_VEL
LIN {X 0,Y 221.828,Z 500.56,A -85,B 0,C 180,E1 -22014.675,E2 -22014.675} C_VEL
LIN {X 0,Y 214.938,Z 507.102,A -85,B 0,C 180,E1 -22017.349,E2 -22017.349} C_VEL
LIN {X 0,Y 209.467,Z 511.725,A -85,B 0,C 180,E1 -22019.782,E2 -22019.782} C_VEL
LIN {X 0,Y 203.357,Z 516.479,A -85,B 0,C 180,E1 -22023.302,E2 -22023.302} C_VEL
LIN {X 0,Y 198.41,Z 519.823,A -85,B 0,C 180,E1 -22027.068,E2 -22027.068} C_VEL
LIN {X 0,Y 194.749,Z 521.849,A -85,B 0,C 180,E1 -22031.047,E2 -22031.047} C_VEL
LIN {X 0,Y 192.393,Z 522.539,A -85,B 0,C 180,E1 -22035.184,E2 -22035.184} C_VEL
LIN {X 0,Y 191.434,Z 521.997,A -85,B 0,C 180,E1 -22039.422,E2 -22039.422} C_VEL
LIN {X 0,Y 191.71,Z 520.029,A -85,B 0,C 180,E1 -22043.685,E2 -22043.685} C_VEL
LIN {X 0,Y 192.785,Z 516.575,A -85,B 0,C 180,E1 -22047.91,E2 -22047.91} C_VEL
LIN {X 0,Y 193.226,Z 513.992,A -85,B 0,C 180,E1 -22050,E2 -22050} C_VEL
LIN {X 0,Y 193.31,Z 510.759,A -85,B 0,C 180,E1 -22052.083,E2 -22052.083} C_VEL
LIN {X 0,Y 193.285,Z 506.783,A -85,B 0,C 180,E1 -22054.164,E2 -22054.164} C_VEL
LIN {X 0,Y 192.677,Z 503.447,A -85,B 0,C 180,E1 -22055.591,E2 -22055.591} C_VEL
LIN {X 0,Y 191.13,Z 499.698,A -85,B 0,C 180,E1 -22056.891,E2 -22056.891} C_VEL
LIN {X 0,Y 187.041,Z 489.969,A -85,B 0,C 180,E1 -22059.7,E2 -22059.7} C_VEL
LIN {X 0,Y 186.468,Z 485.489,A -85,B 0,C 180,E1 -22060.909,E2 -22060.909} C_VEL
LIN {X 0,Y 186.98,Z 474.588,A -85,B 0,C 180,E1 -22063.586,E2 -22063.586} C_VEL
LIN {X 0,Y 187.223,Z 469.271,A -85,B 0,C 180,E1 -22064.677,E2 -22064.677} C_VEL
LIN {X 0,Y 186.033,Z 457.204,A -85,B 0,C 180,E1 -22066.6,E2 -22066.6} C_VEL
LIN {X 0,Y 185.344,Z 445.203,A -85,B 0,C 180,E1 -22068.081,E2 -22068.081} C_VEL
LIN {X 0,Y 185.317,Z 434.705,A -85,B 0,C 180,E1 -22069.099,E2 -22069.099} C_VEL
LIN {X 0,Y 187.798,Z 421.886,A -85,B 0,C 180,E1 -22077.891,E2 -22077.891} C_VEL
LIN {X 0,Y 189.486,Z 416.545,A -85,B 0,C 180,E1 -22081.453,E2 -22081.453} C_VEL
LIN {X 0,Y 189.25,Z 413.932,A -85,B 0,C 180,E1 -22083.212,E2 -22083.212} C_VEL
LIN {X 0,Y 187.602,Z 406.919,A -85,B 0,C 180,E1 -22088.121,E2 -22088.121} C_VEL
LIN {X 0,Y 185.91,Z 398.694,A -85,B 0,C 180,E1 -22094.089,E2 -22094.089} C_VEL
LIN {X 0,Y 185.614,Z 397.36,A -85,B 0,C 180,E1 -22095.126,E2 -22095.126} C_VEL
LIN {X 0,Y 185.492,Z 397.378,A -85,B 0,C 180,E1 -22099.901,E2 -22099.901} C_VEL
LIN {X 0,Y 185.544,Z 397.371,A -85,B 0,C 180,E1 -22102.696,E2 -22102.696} C_VEL
LIN {X 0,Y 185.541,Z 397.372,A -85,B 0,C 180,E1 -22107.974,E2 -22107.974} C_VEL
LIN {X 0,Y 185.581,Z 397.367,A -85,B 0,C 180,E1 -22110.576,E2 -22110.576} C_VEL
LIN {X 0,Y 185.588,Z 397.363,A -85,B 0,C 180,E1 -22115.383,E2 -22115.383} C_VEL
LIN {X 0,Y 185.608,Z 397.364,A -85,B 0,C 180,E1 -22120.075,E2 -22120.075} C_VEL
LIN {X 0,Y 185.725,Z 397.347,A -85,B 0,C 180,E1 -22124.64,E2 -22124.64} C_VEL
LIN {X 0,Y 185.943,Z 397.322,A -85,B 0,C 180,E1 -22129.328,E2 -22129.328} C_VEL
LIN {X 0,Y 185.97,Z 397.318,A -85,B 0,C 180,E1 -22133.49,E2 -22133.49} C_VEL
LIN {X 0,Y 186.212,Z 397.288,A -85,B 0,C 180,E1 -22137.837,E2 -22137.837} C_VEL
LIN {X 0,Y 186.408,Z 397.261,A -85,B 0,C 180,E1 -22140,E2 -22140} C_VEL
LIN {X 0,Y 185.928,Z 397.324,A -85,B 0,C 180,E1 -22144.336,E2 -22144.336} C_VEL
LIN {X 0,Y 186.03,Z 397.307,A -85,B 0,C 180,E1 -22148.692,E2 -22148.692} C_VEL
LIN {X 0,Y 185.766,Z 397.346,A -85,B 0,C 180,E1 -22153.12,E2 -22153.12} C_VEL
LIN {X 0,Y 185.717,Z 397.348,A -85,B 0,C 180,E1 -22157.622,E2 -22157.622} C_VEL
LIN {X 0,Y 185.601,Z 397.364,A -85,B 0,C 180,E1 -22162.251,E2 -22162.251} C_VEL
LIN {X 0,Y 185.563,Z 397.368,A -85,B 0,C 180,E1 -22167.032,E2 -22167.032} C_VEL
LIN {X 0,Y 185.579,Z 397.368,A -85,B 0,C 180,E1 -22169.493,E2 -22169.493} C_VEL
LIN {X 0,Y 185.5,Z 397.374,A -85,B 0,C 180,E1 -22174.632,E2 -22174.632} C_VEL
LIN {X 0,Y 185.506,Z 397.377,A -85,B 0,C 180,E1 -22177.313,E2 -22177.313} C_VEL
LIN {X 0,Y 185.472,Z 397.382,A -85,B 0,C 180,E1 -22180.725,E2 -22180.725} C_VEL
LIN {X 0,Y 185.482,Z 397.379,A -85,B 0,C 180,E1 -22186.048,E2 -22186.048} C_VEL
LIN {X 0,Y 185.49,Z 397.376,A -85,B 0,C 180,E1 -22189.902,E2 -22189.902} C_VEL
LIN {X 0,Y 185.544,Z 397.371,A -85,B 0,C 180,E1 -22192.696,E2 -22192.696} C_VEL
LIN {X 0,Y 185.546,Z 397.371,A -85,B 0,C 180,E1 -22197.976,E2 -22197.976} C_VEL
LIN {X 0,Y 185.583,Z 397.365,A -85,B 0,C 180,E1 -22200.576,E2 -22200.576} C_VEL
LIN {X 0,Y 185.607,Z 397.363,A -85,B 0,C 180,E1 -22205.386,E2 -22205.386} C_VEL
LIN {X 0,Y 185.712,Z 397.35,A -85,B 0,C 180,E1 -22211.101,E2 -22211.101} C_VEL
LIN {X 0,Y 185.731,Z 397.348,A -85,B 0,C 180,E1 -22214.641,E2 -22214.641} C_VEL
LIN {X 0,Y 185.926,Z 397.323,A -85,B 0,C 180,E1 -22219.36,E2 -22219.36} C_VEL
LIN {X 0,Y 185.963,Z 397.319,A -85,B 0,C 180,E1 -22223.49,E2 -22223.49} C_VEL
LIN {X 0,Y 186.21,Z 397.288,A -85,B 0,C 180,E1 -22227.837,E2 -22227.837} C_VEL
LIN {X 0,Y 186.412,Z 397.266,A -85,B 0,C 180,E1 -22230,E2 -22230} C_VEL
LIN {X 0,Y 185.923,Z 397.322,A -85,B 0,C 180,E1 -22234.336,E2 -22234.336} C_VEL
LIN {X 0,Y 185.986,Z 397.316,A -85,B 0,C 180,E1 -22238.694,E2 -22238.694} C_VEL
LIN {X 0,Y 185.734,Z 397.343,A -85,B 0,C 180,E1 -22243.123,E2 -22243.123} C_VEL
LIN {X 0,Y 185.72,Z 397.352,A -85,B 0,C 180,E1 -22247.622,E2 -22247.622} C_VEL
LIN {X 0,Y 185.603,Z 397.362,A -85,B 0,C 180,E1 -22252.251,E2 -22252.251} C_VEL
LIN {X 0,Y 185.565,Z 397.369,A -85,B 0,C 180,E1 -22257.032,E2 -22257.032} C_VEL
LIN {X 0,Y 185.582,Z 397.365,A -85,B 0,C 180,E1 -22259.493,E2 -22259.493} C_VEL
LIN {X 0,Y 185.522,Z 397.374,A -85,B 0,C 180,E1 -22264.628,E2 -22264.628} C_VEL
LIN {X 0,Y 185.546,Z 397.37,A -85,B 0,C 180,E1 -22267.304,E2 -22267.304} C_VEL
LIN {X 0,Y 185.488,Z 397.377,A -85,B 0,C 180,E1 -22270.73,E2 -22270.73} C_VEL
LIN {X 0,Y 185.484,Z 397.379,A -85,B 0,C 180,E1 -22273.953,E2 -22273.953} C_VEL
LIN {X 0,Y 185.486,Z 397.38,A -85,B 0,C 180,E1 -22279.271,E2 -22279.271} C_VEL
LIN {X 0,Y 185.546,Z 397.372,A -85,B 0,C 180,E1 -22282.696,E2 -22282.696} C_VEL
LIN {X 0,Y 185.945,Z 397.486,A -85,B 0,C 180,E1 -22288.402,E2 -22288.402} C_VEL
LIN {X 0,Y 185.512,Z 400.987,A -85,B 0,C 180,E1 -22291.735,E2 -22291.735} C_VEL
LIN {X 0,Y 184.73,Z 407.321,A -85,B 0,C 180,E1 -22297.638,E2 -22297.638} C_VEL
LIN {X 0,Y 184.215,Z 412.646,A -85,B 0,C 180,E1 -22302.513,E2 -22302.513} C_VEL
LIN {X 0,Y 184.154,Z 418.681,A -85,B 0,C 180,E1 -22307.953,E2 -22307.953} C_VEL
LIN {X 0,Y 185.352,Z 431.663,A -85,B 0,C 180,E1 -22309.58,E2 -22309.58} C_VEL
LIN {X 0,Y 185.623,Z 435.923,A -85,B 0,C 180,E1 -22310.223,E2 -22310.223} C_VEL
LIN {X 0,Y 185.062,Z 447.534,A -85,B 0,C 180,E1 -22312.362,E2 -22312.362} C_VEL
LIN {X 0,Y 184.719,Z 457.996,A -85,B 0,C 180,E1 -22314.816,E2 -22314.816} C_VEL
LIN {X 0,Y 184.253,Z 466.402,A -85,B 0,C 180,E1 -22317.267,E2 -22317.267} C_VEL
LIN {X 0,Y 184.1,Z 475.522,A -85,B 0,C 180,E1 -22320.547,E2 -22320.547} C_VEL
LIN {X 0,Y 184.541,Z 482.729,A -85,B 0,C 180,E1 -22323.821,E2 -22323.821} C_VEL
LIN {X 0,Y 185.888,Z 489.192,A -85,B 0,C 180,E1 -22327.604,E2 -22327.604} C_VEL
LIN {X 0,Y 187.926,Z 493.326,A -85,B 0,C 180,E1 -22330.777,E2 -22330.777} C_VEL
LIN {X 0,Y 189.665,Z 495.384,A -85,B 0,C 180,E1 -22332.846,E2 -22332.846} C_VEL
LIN {X 0,Y 191.755,Z 496.963,A -85,B 0,C 180,E1 -22334.866,E2 -22334.866} C_VEL
LIN {X 0,Y 194.151,Z 498,A -85,B 0,C 180,E1 -22336.833,E2 -22336.833} C_VEL
LIN {X 0,Y 196.819,Z 498.562,A -85,B 0,C 180,E1 -22338.746,E2 -22338.746} C_VEL
LIN {X 0,Y 199.738,Z 498.621,A -85,B 0,C 180,E1 -22340.601,E2 -22340.601} C_VEL
LIN {X 0,Y 202.905,Z 498.202,A -85,B 0,C 180,E1 -22342.396,E2 -22342.396} C_VEL
LIN {X 0,Y 206.3,Z 497.341,A -85,B 0,C 180,E1 -22344.13,E2 -22344.13} C_VEL
LIN {X 0,Y 209.947,Z 495.976,A -85,B 0,C 180,E1 -22345.797,E2 -22345.797} C_VEL
LIN {X 0,Y 213.788,Z 494.143,A -85,B 0,C 180,E1 -22347.402,E2 -22347.402} C_VEL
LIN {X 0,Y 217.015,Z 492.176,A -85,B 0,C 180,E1 -22349.063,E2 -22349.063} C_VEL
LIN {X 0,Y 218.996,Z 490.535,A -85,B 0,C 180,E1 -22350.895,E2 -22350.895} C_VEL
LIN {X 0,Y 220.815,Z 488.924,A -85,B 0,C 180,E1 -22352.756,E2 -22352.756} C_VEL
LIN {X 0,Y 222.348,Z 487.421,A -85,B 0,C 180,E1 -22354.733,E2 -22354.733} C_VEL
LIN {X 0,Y 223.459,Z 486.406,A -85,B 0,C 180,E1 -22356.696,E2 -22356.696} C_VEL
LIN {X 0,Y 224.119,Z 485.954,A -85,B 0,C 180,E1 -22358.842,E2 -22358.842} C_VEL
LIN {X 0,Y 224.822,Z 485.999,A -85,B 0,C 180,E1 -22361.388,E2 -22361.388} C_VEL
LIN {X 0,Y 225.312,Z 487.004,A -85,B 0,C 180,E1 -22364.157,E2 -22364.157} C_VEL
LIN {X 0,Y 225.454,Z 488.844,A -85,B 0,C 180,E1 -22366.701,E2 -22366.701} C_VEL
LIN {X 0,Y 225.55,Z 490.466,A -85,B 0,C 180,E1 -22368.403,E2 -22368.403} C_VEL
LIN {X 0,Y 225.316,Z 491.357,A -85,B 0,C 180,E1 -22369.078,E2 -22369.078} C_VEL
LIN {X 0,Y 222.352,Z 495.317,A -85,B 0,C 180,E1 -22370.79,E2 -22370.79} C_VEL
LIN {X 0,Y 219.103,Z 499.227,A -85,B 0,C 180,E1 -22372.45,E2 -22372.45} C_VEL
LIN {X 0,Y 213.124,Z 504.813,A -85,B 0,C 180,E1 -22374.754,E2 -22374.754} C_VEL
LIN {X 0,Y 205.238,Z 510.997,A -85,B 0,C 180,E1 -22377.942,E2 -22377.942} C_VEL
LIN {X 0,Y 200.138,Z 514.585,A -85,B 0,C 180,E1 -22380.552,E2 -22380.552} C_VEL
LIN {X 0,Y 194.274,Z 518.163,A -85,B 0,C 180,E1 -22384.271,E2 -22384.271} C_VEL
LIN {X 0,Y 189.813,Z 520.42,A -85,B 0,C 180,E1 -22388.268,E2 -22388.268} C_VEL
LIN {X 0,Y 186.661,Z 521.422,A -85,B 0,C 180,E1 -22392.469,E2 -22392.469} C_VEL
LIN {X 0,Y 184.886,Z 521.117,A -85,B 0,C 180,E1 -22396.816,E2 -22396.816} C_VEL
LIN {X 0,Y 184.618,Z 519.309,A -85,B 0,C 180,E1 -22401.795,E2 -22401.795} C_VEL
LIN {X 0,Y 185.317,Z 516.571,A -85,B 0,C 180,E1 -22405.65,E2 -22405.65} C_VEL
LIN {X 0,Y 186.289,Z 513.193,A -85,B 0,C 180,E1 -22408.919,E2 -22408.919} C_VEL
LIN {X 0,Y 186.491,Z 510.13,A -85,B 0,C 180,E1 -22411.079,E2 -22411.079} C_VEL
LIN {X 0,Y 186.496,Z 505.098,A -85,B 0,C 180,E1 -22413.829,E2 -22413.829} C_VEL
LIN {X 0,Y 186.278,Z 498.918,A -85,B 0,C 180,E1 -22416.499,E2 -22416.499} C_VEL
LIN {X 0,Y 186.364,Z 490.081,A -85,B 0,C 180,E1 -22419.563,E2 -22419.563} C_VEL
LIN {X 0,Y 186.468,Z 485.489,A -85,B 0,C 180,E1 -22420.909,E2 -22420.909} C_VEL
LIN {X 0,Y 185.952,Z 480.918,A -85,B 0,C 180,E1 -22422.046,E2 -22422.046} C_VEL
LIN {X 0,Y 184.534,Z 476.099,A -85,B 0,C 180,E1 -22423.044,E2 -22423.044} C_VEL
LIN {X 0,Y 180.843,Z 466.036,A -85,B 0,C 180,E1 -22424.806,E2 -22424.806} C_VEL
LIN {X 0,Y 179.293,Z 458.922,A -85,B 0,C 180,E1 -22425.904,E2 -22425.904} C_VEL
LIN {X 0,Y 178.388,Z 446.07,A -85,B 0,C 180,E1 -22427.629,E2 -22427.629} C_VEL
LIN {X 0,Y 178.268,Z 434.432,A -85,B 0,C 180,E1 -22428.831,E2 -22428.831} C_VEL
LIN {X 0,Y 180.637,Z 421.929,A -85,B 0,C 180,E1 -22437.832,E2 -22437.832} C_VEL
LIN {X 0,Y 182.138,Z 417.274,A -85,B 0,C 180,E1 -22441.094,E2 -22441.094} C_VEL
LIN {X 0,Y 182.359,Z 415.048,A -85,B 0,C 180,E1 -22442.653,E2 -22442.653} C_VEL
LIN {X 0,Y 180.636,Z 407.96,A -85,B 0,C 180,E1 -22447.791,E2 -22447.791} C_VEL
LIN {X 0,Y 179.039,Z 400.517,A -85,B 0,C 180,E1 -22453.431,E2 -22453.431} C_VEL
LIN {X 0,Y 178.556,Z 398.239,A -85,B 0,C 180,E1 -22455.29,E2 -22455.29} C_VEL
LIN {X 0,Y 178.42,Z 398.259,A -85,B 0,C 180,E1 -22460.932,E2 -22460.932} C_VEL
LIN {X 0,Y 178.495,Z 398.247,A -85,B 0,C 180,E1 -22465.776,E2 -22465.776} C_VEL
LIN {X 0,Y 178.522,Z 398.249,A -85,B 0,C 180,E1 -22470.007,E2 -22470.007} C_VEL
LIN {X 0,Y 178.535,Z 398.241,A -85,B 0,C 180,E1 -22474.876,E2 -22474.876} C_VEL
LIN {X 0,Y 178.624,Z 398.232,A -85,B 0,C 180,E1 -22480.784,E2 -22480.784} C_VEL
LIN {X 0,Y 178.666,Z 398.228,A -85,B 0,C 180,E1 -22484.017,E2 -22484.017} C_VEL
LIN {X 0,Y 178.895,Z 398.2,A -85,B 0,C 180,E1 -22489.153,E2 -22489.153} C_VEL
LIN {X 0,Y 178.935,Z 398.193,A -85,B 0,C 180,E1 -22493.233,E2 -22493.233} C_VEL
LIN {X 0,Y 179.157,Z 398.167,A -85,B 0,C 180,E1 -22497.752,E2 -22497.752} C_VEL
LIN {X 0,Y 179.371,Z 398.137,A -85,B 0,C 180,E1 -22500,E2 -22500} C_VEL
LIN {X 0,Y 178.877,Z 398.202,A -85,B 0,C 180,E1 -22504.507,E2 -22504.507} C_VEL
LIN {X 0,Y 178.979,Z 398.186,A -85,B 0,C 180,E1 -22509.037,E2 -22509.037} C_VEL
LIN {X 0,Y 178.689,Z 398.226,A -85,B 0,C 180,E1 -22513.65,E2 -22513.65} C_VEL
LIN {X 0,Y 178.671,Z 398.225,A -85,B 0,C 180,E1 -22518.342,E2 -22518.342} C_VEL
LIN {X 0,Y 178.514,Z 398.248,A -85,B 0,C 180,E1 -22523.185,E2 -22523.185} C_VEL
LIN {X 0,Y 178.488,Z 398.249,A -85,B 0,C 180,E1 -22528.197,E2 -22528.197} C_VEL
LIN {X 0,Y 178.501,Z 398.251,A -85,B 0,C 180,E1 -22530.787,E2 -22530.787} C_VEL
LIN {X 0,Y 178.485,Z 398.246,A -85,B 0,C 180,E1 -22534.22,E2 -22534.22} C_VEL
LIN {X 0,Y 178.396,Z 398.263,A -85,B 0,C 180,E1 -22539.074,E2 -22539.074} C_VEL
LIN {X 0,Y 178.399,Z 398.259,A -85,B 0,C 180,E1 -22542.045,E2 -22542.045} C_VEL
LIN {X 0,Y 178.403,Z 398.261,A -85,B 0,C 180,E1 -22545.161,E2 -22545.161} C_VEL
LIN {X 0,Y 178.416,Z 398.261,A -85,B 0,C 180,E1 -22548.455,E2 -22548.455} C_VEL
LIN {X 0,Y 178.465,Z 398.249,A -85,B 0,C 180,E1 -22551.963,E2 -22551.963} C_VEL
LIN {X 0,Y 178.492,Z 398.252,A -85,B 0,C 180,E1 -22556.548,E2 -22556.548} C_VEL
LIN {X 0,Y 178.524,Z 398.243,A -85,B 0,C 180,E1 -22560.007,E2 -22560.007} C_VEL
LIN {X 0,Y 178.536,Z 398.245,A -85,B 0,C 180,E1 -22564.876,E2 -22564.876} C_VEL
LIN {X 0,Y 178.656,Z 398.23,A -85,B 0,C 180,E1 -22570.755,E2 -22570.755} C_VEL
LIN {X 0,Y 178.678,Z 398.229,A -85,B 0,C 180,E1 -22574.019,E2 -22574.019} C_VEL
LIN {X 0,Y 178.863,Z 398.202,A -85,B 0,C 180,E1 -22579.21,E2 -22579.21} C_VEL
LIN {X 0,Y 178.927,Z 398.195,A -85,B 0,C 180,E1 -22583.233,E2 -22583.233} C_VEL
LIN {X 0,Y 179.156,Z 398.166,A -85,B 0,C 180,E1 -22587.752,E2 -22587.752} C_VEL
LIN {X 0,Y 179.375,Z 398.143,A -85,B 0,C 180,E1 -22590,E2 -22590} C_VEL
LIN {X 0,Y 178.87,Z 398.199,A -85,B 0,C 180,E1 -22594.508,E2 -22594.508} C_VEL
LIN {X 0,Y 178.914,Z 398.197,A -85,B 0,C 180,E1 -22599.041,E2 -22599.041} C_VEL
LIN {X 0,Y 178.662,Z 398.226,A -85,B 0,C 180,E1 -22603.652,E2 -22603.652} C_VEL
LIN {X 0,Y 178.641,Z 398.232,A -85,B 0,C 180,E1 -22609.231,E2 -22609.231} C_VEL
LIN {X 0,Y 178.537,Z 398.245,A -85,B 0,C 180,E1 -22615.125,E2 -22615.125} C_VEL
LIN {X 0,Y 178.482,Z 398.247,A -85,B 0,C 180,E1 -22620.791,E2 -22620.791} C_VEL
LIN {X 0,Y 178.499,Z 398.249,A -85,B 0,C 180,E1 -22624.225,E2 -22624.225} C_VEL
LIN {X 0,Y 178.421,Z 398.255,A -85,B 0,C 180,E1 -22629.069,E2 -22629.069} C_VEL
LIN {X 0,Y 178.414,Z 398.26,A -85,B 0,C 180,E1 -22632.041,E2 -22632.041} C_VEL
LIN {X 0,Y 178.402,Z 398.262,A -85,B 0,C 180,E1 -22635.162,E2 -22635.162} C_VEL
LIN {X 0,Y 178.412,Z 398.257,A -85,B 0,C 180,E1 -22638.457,E2 -22638.457} C_VEL
LIN {X 0,Y 178.52,Z 398.245,A -85,B 0,C 180,E1 -22643.806,E2 -22643.806} C_VEL
LIN {X 0,Y 178.878,Z 398.267,A -85,B 0,C 180,E1 -22648.464,E2 -22648.464} C_VEL
LIN {X 0,Y 178.224,Z 402.932,A -85,B 0,C 180,E1 -22653.032,E2 -22653.032} C_VEL
LIN {X 0,Y 177.617,Z 408.04,A -85,B 0,C 180,E1 -22657.92,E2 -22657.92} C_VEL
LIN {X 0,Y 177.158,Z 412.554,A -85,B 0,C 180,E1 -22662.196,E2 -22662.196} C_VEL
LIN {X 0,Y 177.084,Z 418.995,A -85,B 0,C 180,E1 -22668.192,E2 -22668.192} C_VEL
LIN {X 0,Y 178.417,Z 432.525,A -85,B 0,C 180,E1 -22669.992,E2 -22669.992} C_VEL
LIN {X 0,Y 178.438,Z 438.216,A -85,B 0,C 180,E1 -22670.936,E2 -22670.936} C_VEL
LIN {X 0,Y 177.927,Z 449.402,A -85,B 0,C 180,E1 -22673.195,E2 -22673.195} C_VEL
LIN {X 0,Y 177.605,Z 459.55,A -85,B 0,C 180,E1 -22675.745,E2 -22675.745} C_VEL
LIN {X 0,Y 177.163,Z 467.806,A -85,B 0,C 180,E1 -22678.295,E2 -22678.295} C_VEL
LIN {X 0,Y 177.129,Z 475.346,A -85,B 0,C 180,E1 -22681.137,E2 -22681.137} C_VEL
LIN {X 0,Y 177.659,Z 482.696,A -85,B 0,C 180,E1 -22684.538,E2 -22684.538} C_VEL
LIN {X 0,Y 178.888,Z 488.543,A -85,B 0,C 180,E1 -22687.903,E2 -22687.903} C_VEL
LIN {X 0,Y 180.955,Z 493.049,A -85,B 0,C 180,E1 -22691.198,E2 -22691.198} C_VEL
LIN {X 0,Y 182.756,Z 495.368,A -85,B 0,C 180,E1 -22693.34,E2 -22693.34} C_VEL
LIN {X 0,Y 184.899,Z 497.193,A -85,B 0,C 180,E1 -22695.43,E2 -22695.43} C_VEL
LIN {X 0,Y 187.373,Z 498.502,A -85,B 0,C 180,E1 -22697.462,E2 -22697.462} C_VEL
LIN {X 0,Y 190.16,Z 499.318,A -85,B 0,C 180,E1 -22699.428,E2 -22699.428} C_VEL
LIN {X 0,Y 193.173,Z 499.669,A -85,B 0,C 180,E1 -22701.335,E2 -22701.335} C_VEL
LIN {X 0,Y 196.442,Z 499.53,A -85,B 0,C 180,E1 -22703.175,E2 -22703.175} C_VEL
LIN {X 0,Y 199.971,Z 498.955,A -85,B 0,C 180,E1 -22704.945,E2 -22704.945} C_VEL
LIN {X 0,Y 207.717,Z 496.382,A -85,B 0,C 180,E1 -22708.274,E2 -22708.274} C_VEL
LIN {X 0,Y 211.166,Z 494.674,A -85,B 0,C 180,E1 -22709.949,E2 -22709.949} C_VEL
LIN {X 0,Y 213.319,Z 493.309,A -85,B 0,C 180,E1 -22711.812,E2 -22711.812} C_VEL
LIN {X 0,Y 215.252,Z 491.991,A -85,B 0,C 180,E1 -22713.714,E2 -22713.714} C_VEL
LIN {X 0,Y 216.967,Z 490.803,A -85,B 0,C 180,E1 -22715.923,E2 -22715.923} C_VEL
LIN {X 0,Y 217.907,Z 490.198,A -85,B 0,C 180,E1 -22717.792,E2 -22717.792} C_VEL
LIN {X 0,Y 218.654,Z 490.127,A -85,B 0,C 180,E1 -22720.004,E2 -22720.004} C_VEL
LIN {X 0,Y 219.327,Z 490.554,A -85,B 0,C 180,E1 -22722.523,E2 -22722.523} C_VEL
LIN {X 0,Y 219.59,Z 491.956,A -85,B 0,C 180,E1 -22725.241,E2 -22725.241} C_VEL
LIN {X 0,Y 219.631,Z 493.969,A -85,B 0,C 180,E1 -22727.779,E2 -22727.779} C_VEL
LIN {X 0,Y 218.74,Z 495.495,A -85,B 0,C 180,E1 -22728.802,E2 -22728.802} C_VEL
LIN {X 0,Y 213.675,Z 500.868,A -85,B 0,C 180,E1 -22731.322,E2 -22731.322} C_VEL
LIN {X 0,Y 207.423,Z 506.003,A -85,B 0,C 180,E1 -22733.633,E2 -22733.633} C_VEL
LIN {X 0,Y 199.282,Z 511.568,A -85,B 0,C 180,E1 -22736.863,E2 -22736.863} C_VEL
LIN {X 0,Y 193.991,Z 514.776,A -85,B 0,C 180,E1 -22739.522,E2 -22739.522} C_VEL
LIN {X 0,Y 187.913,Z 517.902,A -85,B 0,C 180,E1 -22743.333,E2 -22743.333} C_VEL
LIN {X 0,Y 183.249,Z 519.727,A -85,B 0,C 180,E1 -22747.447,E2 -22747.447} C_VEL
LIN {X 0,Y 179.923,Z 520.337,A -85,B 0,C 180,E1 -22751.79,E2 -22751.79} C_VEL
LIN {X 0,Y 178.056,Z 519.718,A -85,B 0,C 180,E1 -22756.3,E2 -22756.3} C_VEL
LIN {X 0,Y 177.76,Z 517.629,A -85,B 0,C 180,E1 -22761.271,E2 -22761.271} C_VEL
LIN {X 0,Y 178.5,Z 514.566,A -85,B 0,C 180,E1 -22765.483,E2 -22765.483} C_VEL
LIN {X 0,Y 179.557,Z 510.9,A -85,B 0,C 180,E1 -22768.878,E2 -22768.878} C_VEL
LIN {X 0,Y 179.76,Z 507.556,A -85,B 0,C 180,E1 -22771.12,E2 -22771.12} C_VEL
LIN {X 0,Y 179.746,Z 502.32,A -85,B 0,C 180,E1 -22773.923,E2 -22773.923} C_VEL
LIN {X 0,Y 179.444,Z 495.636,A -85,B 0,C 180,E1 -22776.747,E2 -22776.747} C_VEL
LIN {X 0,Y 179.54,Z 487.606,A -85,B 0,C 180,E1 -22779.511,E2 -22779.511} C_VEL
LIN {X 0,Y 179.812,Z 477.524,A -85,B 0,C 180,E1 -22782.277,E2 -22782.277} C_VEL
LIN {X 0,Y 180.295,Z 469.422,A -85,B 0,C 180,E1 -22784.1,E2 -22784.1} C_VEL
LIN {X 0,Y 179.293,Z 458.922,A -85,B 0,C 180,E1 -22785.904,E2 -22785.904} C_VEL
LIN {X 0,Y 178.31,Z 455.372,A -85,B 0,C 180,E1 -22786.391,E2 -22786.391} C_VEL
LIN {X 0,Y 171.98,Z 443.931,A -85,B 0,C 180,E1 -22787.534,E2 -22787.534} C_VEL
LIN {X 0,Y 171.211,Z 440.189,A -85,B 0,C 180,E1 -22787.904,E2 -22787.904} C_VEL
LIN {X 0,Y 171.233,Z 434.042,A -85,B 0,C 180,E1 -22788.547,E2 -22788.547} C_VEL
LIN {X 0,Y 173.463,Z 421.91,A -85,B 0,C 180,E1 -22797.769,E2 -22797.769} C_VEL
LIN {X 0,Y 175.124,Z 416.928,A -85,B 0,C 180,E1 -22801.447,E2 -22801.447} C_VEL
LIN {X 0,Y 175.253,Z 415.318,A -85,B 0,C 180,E1 -22802.633,E2 -22802.633} C_VEL
LIN {X 0,Y 173.697,Z 409.071,A -85,B 0,C 180,E1 -22807.366,E2 -22807.366} C_VEL
LIN {X 0,Y 172.178,Z 402.258,A -85,B 0,C 180,E1 -22812.716,E2 -22812.716} C_VEL
LIN {X 0,Y 171.512,Z 399.117,A -85,B 0,C 180,E1 -22815.377,E2 -22815.377} C_VEL
LIN {X 0,Y 171.414,Z 399.134,A -85,B 0,C 180,E1 -22822.048,E2 -22822.048} C_VEL
LIN {X 0,Y 171.41,Z 399.128,A -85,B 0,C 180,E1 -22825.087,E2 -22825.087} C_VEL
LIN {X 0,Y 171.448,Z 399.128,A -85,B 0,C 180,E1 -22830.534,E2 -22830.534} C_VEL
LIN {X 0,Y 171.458,Z 399.125,A -85,B 0,C 180,E1 -22835.802,E2 -22835.802} C_VEL
LIN {X 0,Y 171.58,Z 399.109,A -85,B 0,C 180,E1 -22840.872,E2 -22840.872} C_VEL
LIN {X 0,Y 171.61,Z 399.109,A -85,B 0,C 180,E1 -22845.776,E2 -22845.776} C_VEL
LIN {X 0,Y 171.911,Z 399.066,A -85,B 0,C 180,E1 -22850.588,E2 -22850.588} C_VEL
LIN {X 0,Y 171.829,Z 399.081,A -85,B 0,C 180,E1 -22855.308,E2 -22855.308} C_VEL
LIN {X 0,Y 172.334,Z 399.013,A -85,B 0,C 180,E1 -22860,E2 -22860} C_VEL
LIN {X 0,Y 171.826,Z 399.081,A -85,B 0,C 180,E1 -22864.692,E2 -22864.692} C_VEL
LIN {X 0,Y 171.911,Z 399.067,A -85,B 0,C 180,E1 -22869.412,E2 -22869.412} C_VEL
LIN {X 0,Y 171.614,Z 399.106,A -85,B 0,C 180,E1 -22874.224,E2 -22874.224} C_VEL
LIN {X 0,Y 171.558,Z 399.114,A -85,B 0,C 180,E1 -22879.575,E2 -22879.575} C_VEL
LIN {X 0,Y 171.47,Z 399.121,A -85,B 0,C 180,E1 -22885.617,E2 -22885.617} C_VEL
LIN {X 0,Y 171.459,Z 399.127,A -85,B 0,C 180,E1 -22890.597,E2 -22890.597} C_VEL
LIN {X 0,Y 171.393,Z 399.132,A -85,B 0,C 180,E1 -22895.035,E2 -22895.035} C_VEL
LIN {X 0,Y 171.358,Z 399.141,A -85,B 0,C 180,E1 -22898.808,E2 -22898.808} C_VEL
LIN {X 0,Y 171.326,Z 399.14,A -85,B 0,C 180,E1 -22904.216,E2 -22904.216} C_VEL
LIN {X 0,Y 171.349,Z 399.139,A -85,B 0,C 180,E1 -22908.986,E2 -22908.986} C_VEL
LIN {X 0,Y 171.414,Z 399.127,A -85,B 0,C 180,E1 -22912.048,E2 -22912.048} C_VEL
LIN {X 0,Y 171.412,Z 399.133,A -85,B 0,C 180,E1 -22915.087,E2 -22915.087} C_VEL
LIN {X 0,Y 171.451,Z 399.124,A -85,B 0,C 180,E1 -22920.535,E2 -22920.535} C_VEL
LIN {X 0,Y 171.467,Z 399.125,A -85,B 0,C 180,E1 -22925.804,E2 -22925.804} C_VEL
LIN {X 0,Y 171.612,Z 399.107,A -85,B 0,C 180,E1 -22930.876,E2 -22930.876} C_VEL
LIN {X 0,Y 171.615,Z 399.106,A -85,B 0,C 180,E1 -22935.776,E2 -22935.776} C_VEL
LIN {X 0,Y 171.891,Z 399.073,A -85,B 0,C 180,E1 -22940.588,E2 -22940.588} C_VEL
LIN {X 0,Y 171.824,Z 399.077,A -85,B 0,C 180,E1 -22945.308,E2 -22945.308} C_VEL
LIN {X 0,Y 172.337,Z 399.019,A -85,B 0,C 180,E1 -22950,E2 -22950} C_VEL
LIN {X 0,Y 171.819,Z 399.077,A -85,B 0,C 180,E1 -22954.693,E2 -22954.693} C_VEL
LIN {X 0,Y 171.85,Z 399.078,A -85,B 0,C 180,E1 -22959.415,E2 -22959.415} C_VEL
LIN {X 0,Y 171.583,Z 399.11,A -85,B 0,C 180,E1 -22964.227,E2 -22964.227} C_VEL
LIN {X 0,Y 171.56,Z 399.113,A -85,B 0,C 180,E1 -22969.575,E2 -22969.575} C_VEL
LIN {X 0,Y 171.472,Z 399.127,A -85,B 0,C 180,E1 -22975.617,E2 -22975.617} C_VEL
LIN {X 0,Y 171.444,Z 399.123,A -85,B 0,C 180,E1 -22980.587,E2 -22980.587} C_VEL
LIN {X 0,Y 171.409,Z 399.133,A -85,B 0,C 180,E1 -22985.032,E2 -22985.032} C_VEL
LIN {X 0,Y 171.382,Z 399.131,A -85,B 0,C 180,E1 -22988.817,E2 -22988.817} C_VEL
LIN {X 0,Y 171.332,Z 399.141,A -85,B 0,C 180,E1 -22994.214,E2 -22994.214} C_VEL
LIN {X 0,Y 171.346,Z 399.139,A -85,B 0,C 180,E1 -22998.984,E2 -22998.984} C_VEL
LIN {X 0,Y 171.42,Z 399.131,A -85,B 0,C 180,E1 -23002.049,E2 -23002.049} C_VEL
LIN {X 0,Y 171.829,Z 399.073,A -85,B 0,C 180,E1 -23007.879,E2 -23007.879} C_VEL
LIN {X 0,Y 171.814,Z 399.175,A -85,B 0,C 180,E1 -23008.678,E2 -23008.678} C_VEL
LIN {X 0,Y 171.123,Z 403.595,A -85,B 0,C 180,E1 -23013.143,E2 -23013.143} C_VEL
LIN {X 0,Y 170.471,Z 408.712,A -85,B 0,C 180,E1 -23018.22,E2 -23018.22} C_VEL
LIN {X 0,Y 169.969,Z 413.779,A -85,B 0,C 180,E1 -23023.175,E2 -23023.175} C_VEL
LIN {X 0,Y 170.13,Z 419.565,A -85,B 0,C 180,E1 -23028.625,E2 -23028.625} C_VEL
LIN {X 0,Y 171.396,Z 432.206,A -85,B 0,C 180,E1 -23030.326,E2 -23030.326} C_VEL
LIN {X 0,Y 171.378,Z 438.761,A -85,B 0,C 180,E1 -23031.451,E2 -23031.451} C_VEL
LIN {X 0,Y 170.904,Z 449.953,A -85,B 0,C 180,E1 -23033.803,E2 -23033.803} C_VEL
LIN {X 0,Y 170.585,Z 459.08,A -85,B 0,C 180,E1 -23036.161,E2 -23036.161} C_VEL
LIN {X 0,Y 170.175,Z 469.002,A -85,B 0,C 180,E1 -23039.408,E2 -23039.408} C_VEL
LIN {X 0,Y 170.347,Z 477.764,A -85,B 0,C 180,E1 -23042.956,E2 -23042.956} C_VEL
LIN {X 0,Y 170.99,Z 483.706,A -85,B 0,C 180,E1 -23045.898,E2 -23045.898} C_VEL
LIN {X 0,Y 172.49,Z 489.448,A -85,B 0,C 180,E1 -23049.38,E2 -23049.38} C_VEL
LIN {X 0,Y 174.914,Z 493.984,A -85,B 0,C 180,E1 -23052.767,E2 -23052.767} C_VEL
LIN {X 0,Y 178.067,Z 497.25,A -85,B 0,C 180,E1 -23056.038,E2 -23056.038} C_VEL
LIN {X 0,Y 180.61,Z 498.851,A -85,B 0,C 180,E1 -23058.138,E2 -23058.138} C_VEL
LIN {X 0,Y 183.505,Z 499.928,A -85,B 0,C 180,E1 -23060.163,E2 -23060.163} C_VEL
LIN {X 0,Y 186.623,Z 500.566,A -85,B 0,C 180,E1 -23062.123,E2 -23062.123} C_VEL
LIN {X 0,Y 190.011,Z 500.697,A -85,B 0,C 180,E1 -23064.008,E2 -23064.008} C_VEL
LIN {X 0,Y 193.667,Z 500.401,A -85,B 0,C 180,E1 -23065.815,E2 -23065.815} C_VEL
LIN {X 0,Y 199.975,Z 498.974,A -85,B 0,C 180,E1 -23068.524,E2 -23068.524} C_VEL
LIN {X 0,Y 201.677,Z 498.443,A -85,B 0,C 180,E1 -23069.201,E2 -23069.201} C_VEL
LIN {X 0,Y 205.316,Z 497.011,A -85,B 0,C 180,E1 -23070.894,E2 -23070.894} C_VEL
LIN {X 0,Y 207.599,Z 495.954,A -85,B 0,C 180,E1 -23072.797,E2 -23072.797} C_VEL
LIN {X 0,Y 209.607,Z 494.927,A -85,B 0,C 180,E1 -23074.75,E2 -23074.75} C_VEL
LIN {X 0,Y 211.33,Z 494.126,A -85,B 0,C 180,E1 -23077.046,E2 -23077.046} C_VEL
LIN {X 0,Y 212.272,Z 493.911,A -85,B 0,C 180,E1 -23078.981,E2 -23078.981} C_VEL
LIN {X 0,Y 212.989,Z 494.123,A -85,B 0,C 180,E1 -23081.295,E2 -23081.295} C_VEL
LIN {X 0,Y 213.436,Z 494.978,A -85,B 0,C 180,E1 -23083.748,E2 -23083.748} C_VEL
LIN {X 0,Y 213.536,Z 497.102,A -85,B 0,C 180,E1 -23087.079,E2 -23087.079} C_VEL
LIN {X 0,Y 213.037,Z 497.992,A -85,B 0,C 180,E1 -23087.841,E2 -23087.841} C_VEL
LIN {X 0,Y 208.305,Z 502.382,A -85,B 0,C 180,E1 -23090.13,E2 -23090.13} C_VEL
LIN {X 0,Y 201.805,Z 507.027,A -85,B 0,C 180,E1 -23092.45,E2 -23092.45} C_VEL
LIN {X 0,Y 193.406,Z 512.011,A -85,B 0,C 180,E1 -23095.719,E2 -23095.719} C_VEL
LIN {X 0,Y 187.92,Z 514.837,A -85,B 0,C 180,E1 -23098.426,E2 -23098.426} C_VEL
LIN {X 0,Y 181.592,Z 517.5,A -85,B 0,C 180,E1 -23102.326,E2 -23102.326} C_VEL
LIN {X 0,Y 176.726,Z 518.908,A -85,B 0,C 180,E1 -23106.566,E2 -23106.566} C_VEL
LIN {X 0,Y 173.237,Z 519.126,A -85,B 0,C 180,E1 -23111.061,E2 -23111.061} C_VEL
LIN {X 0,Y 171.274,Z 518.156,A -85,B 0,C 180,E1 -23115.747,E2 -23115.747} C_VEL
LIN {X 0,Y 170.905,Z 515.836,A -85,B 0,C 180,E1 -23120.728,E2 -23120.728} C_VEL
LIN {X 0,Y 171.77,Z 512.337,A -85,B 0,C 180,E1 -23125.306,E2 -23125.306} C_VEL
LIN {X 0,Y 172.574,Z 509.93,A -85,B 0,C 180,E1 -23127.666,E2 -23127.666} C_VEL
LIN {X 0,Y 172.998,Z 506.774,A -85,B 0,C 180,E1 -23130,E2 -23130} C_VEL
LIN {X 0,Y 173.038,Z 501.648,A -85,B 0,C 180,E1 -23132.91,E2 -23132.91} C_VEL
LIN {X 0,Y 172.742,Z 495.071,A -85,B 0,C 180,E1 -23135.837,E2 -23135.837} C_VEL
LIN {X 0,Y 172.746,Z 486.982,A -85,B 0,C 180,E1 -23138.775,E2 -23138.775} C_VEL
LIN {X 0,Y 172.928,Z 476.801,A -85,B 0,C 180,E1 -23141.724,E2 -23141.724} C_VEL
LIN {X 0,Y 173.361,Z 468.09,A -85,B 0,C 180,E1 -23143.776,E2 -23143.776} C_VEL
LIN {X 0,Y 172.038,Z 456.083,A -85,B 0,C 180,E1 -23145.854,E2 -23145.854} C_VEL
LIN {X 0,Y 171.317,Z 444.198,A -85,B 0,C 180,E1 -23147.456,E2 -23147.456} C_VEL
LIN {X 0,Y 171.211,Z 440.189,A -85,B 0,C 180,E1 -23147.904,E2 -23147.904} C_VEL
LIN {X 0,Y 170.829,Z 436.902,A -85,B 0,C 180,E1 -23148.459,E2 -23148.459} C_VEL
LIN {X 0,Y 169.768,Z 433.576,A -85,B 0,C 180,E1 -23149.519,E2 -23149.519} C_VEL
LIN {X 0,Y 167.939,Z 430.074,A -85,B 0,C 180,E1 -23151.38,E2 -23151.38} C_VEL
LIN {X 0,Y 166.124,Z 426.632,A -85,B 0,C 180,E1 -23153.965,E2 -23153.965} C_VEL
LIN {X 0,Y 165.74,Z 424.051,A -85,B 0,C 180,E1 -23155.978,E2 -23155.978} C_VEL
LIN {X 0,Y 165.896,Z 423.197,A -85,B 0,C 180,E1 -23156.649,E2 -23156.649} C_VEL
LIN {X 0,Y 167.983,Z 416.956,A -85,B 0,C 180,E1 -23161.531,E2 -23161.531} C_VEL
LIN {X 0,Y 167.917,Z 414.839,A -85,B 0,C 180,E1 -23163.166,E2 -23163.166} C_VEL
LIN {X 0,Y 166.001,Z 407.024,A -85,B 0,C 180,E1 -23169.424,E2 -23169.424} C_VEL
LIN {X 0,Y 164.47,Z 399.994,A -85,B 0,C 180,E1 -23175.372,E2 -23175.372} C_VEL
LIN {X 0,Y 164.307,Z 400.019,A -85,B 0,C 180,E1 -23180.346,E2 -23180.346} C_VEL
LIN {X 0,Y 164.343,Z 400.01,A -85,B 0,C 180,E1 -23184.342,E2 -23184.342} C_VEL
LIN {X 0,Y 164.389,Z 400.007,A -85,B 0,C 180,E1 -23189.134,E2 -23189.134} C_VEL
LIN {X 0,Y 164.416,Z 399.999,A -85,B 0,C 180,E1 -23194.694,E2 -23194.694} C_VEL
LIN {X 0,Y 164.485,Z 399.995,A -85,B 0,C 180,E1 -23200.051,E2 -23200.051} C_VEL
LIN {X 0,Y 164.554,Z 399.985,A -85,B 0,C 180,E1 -23205.152,E2 -23205.152} C_VEL
LIN {X 0,Y 164.853,Z 399.946,A -85,B 0,C 180,E1 -23210.182,E2 -23210.182} C_VEL
LIN {X 0,Y 164.779,Z 399.959,A -85,B 0,C 180,E1 -23215.107,E2 -23215.107} C_VEL
LIN {X 0,Y 165.297,Z 399.89,A -85,B 0,C 180,E1 -23220,E2 -23220} C_VEL
LIN {X 0,Y 164.842,Z 399.947,A -85,B 0,C 180,E1 -23227.115,E2 -23227.115} C_VEL
LIN {X 0,Y 164.78,Z 399.958,A -85,B 0,C 180,E1 -23231.198,E2 -23231.198} C_VEL
LIN {X 0,Y 164.52,Z 399.987,A -85,B 0,C 180,E1 -23237.399,E2 -23237.399} C_VEL
LIN {X 0,Y 164.475,Z 399.996,A -85,B 0,C 180,E1 -23239.989,E2 -23239.989} C_VEL
LIN {X 0,Y 164.394,Z 400.001,A -85,B 0,C 180,E1 -23246.134,E2 -23246.134} C_VEL
LIN {X 0,Y 164.389,Z 400.007,A -85,B 0,C 180,E1 -23251.236,E2 -23251.236} C_VEL
LIN {X 0,Y 164.295,Z 400.019,A -85,B 0,C 180,E1 -23256.79,E2 -23256.79} C_VEL
LIN {X 0,Y 164.291,Z 400.018,A -85,B 0,C 180,E1 -23259.916,E2 -23259.916} C_VEL
LIN {X 0,Y 164.279,Z 400.017,A -85,B 0,C 180,E1 -23263.342,E2 -23263.342} C_VEL
LIN {X 0,Y 164.292,Z 400.021,A -85,B 0,C 180,E1 -23266.809,E2 -23266.809} C_VEL
LIN {X 0,Y 164.307,Z 400.016,A -85,B 0,C 180,E1 -23270.348,E2 -23270.348} C_VEL
LIN {X 0,Y 164.344,Z 400.013,A -85,B 0,C 180,E1 -23274.343,E2 -23274.343} C_VEL
LIN {X 0,Y 164.392,Z 400.002,A -85,B 0,C 180,E1 -23279.135,E2 -23279.135} C_VEL
LIN {X 0,Y 164.42,Z 400.004,A -85,B 0,C 180,E1 -23284.695,E2 -23284.695} C_VEL
LIN {X 0,Y 164.521,Z 399.988,A -85,B 0,C 180,E1 -23290.017,E2 -23290.017} C_VEL
LIN {X 0,Y 164.561,Z 399.983,A -85,B 0,C 180,E1 -23295.153,E2 -23295.153} C_VEL
LIN {X 0,Y 164.811,Z 399.956,A -85,B 0,C 180,E1 -23300.179,E2 -23300.179} C_VEL
LIN {X 0,Y 164.853,Z 399.949,A -85,B 0,C 180,E1 -23302.652,E2 -23302.652} C_VEL
LIN {X 0,Y 165.052,Z 399.922,A -85,B 0,C 180,E1 -23307.56,E2 -23307.56} C_VEL
LIN {X 0,Y 165.3,Z 399.896,A -85,B 0,C 180,E1 -23310,E2 -23310} C_VEL
LIN {X 0,Y 164.767,Z 399.955,A -85,B 0,C 180,E1 -23314.894,E2 -23314.894} C_VEL
LIN {X 0,Y 164.834,Z 399.951,A -85,B 0,C 180,E1 -23317.349,E2 -23317.349} C_VEL
LIN {X 0,Y 164.705,Z 399.966,A -85,B 0,C 180,E1 -23321.062,E2 -23321.062} C_VEL
LIN {X 0,Y 164.501,Z 399.994,A -85,B 0,C 180,E1 -23327.402,E2 -23327.402} C_VEL
LIN {X 0,Y 164.477,Z 399.993,A -85,B 0,C 180,E1 -23329.989,E2 -23329.989} C_VEL
LIN {X 0,Y 164.396,Z 400.006,A -85,B 0,C 180,E1 -23336.134,E2 -23336.134} C_VEL
LIN {X 0,Y 164.378,Z 400.005,A -85,B 0,C 180,E1 -23341.229,E2 -23341.229} C_VEL
LIN {X 0,Y 164.315,Z 400.015,A -85,B 0,C 180,E1 -23346.785,E2 -23346.785} C_VEL
LIN {X 0,Y 164.303,Z 400.016,A -85,B 0,C 180,E1 -23349.913,E2 -23349.913} C_VEL
LIN {X 0,Y 164.281,Z 400.022,A -85,B 0,C 180,E1 -23353.342,E2 -23353.342} C_VEL
LIN {X 0,Y 164.294,Z 400.016,A -85,B 0,C 180,E1 -23356.809,E2 -23356.809} C_VEL
LIN {X 0,Y 164.307,Z 400.017,A -85,B 0,C 180,E1 -23360.348,E2 -23360.348} C_VEL
LIN {X 0,Y 164.582,Z 399.976,A -85,B 0,C 180,E1 -23366.28,E2 -23366.28} C_VEL
LIN {X 0,Y 164.681,Z 400.127,A -85,B 0,C 180,E1 -23368.978,E2 -23368.978} C_VEL
LIN {X 0,Y 163.85,Z 405.199,A -85,B 0,C 180,E1 -23374.258,E2 -23374.258} C_VEL
LIN {X 0,Y 163.199,Z 410.64,A -85,B 0,C 180,E1 -23379.848,E2 -23379.848} C_VEL
LIN {X 0,Y 162.7,Z 416.998,A -85,B 0,C 180,E1 -23386.256,E2 -23386.256} C_VEL
LIN {X 0,Y 163.115,Z 419.72,A -85,B 0,C 180,E1 -23388.977,E2 -23388.977} C_VEL
LIN {X 0,Y 164.544,Z 434.36,A -85,B 0,C 180,E1 -23391.093,E2 -23391.093} C_VEL
LIN {X 0,Y 164.084,Z 445.166,A -85,B 0,C 180,E1 -23393.236,E2 -23393.236} C_VEL
LIN {X 0,Y 163.755,Z 456.183,A -85,B 0,C 180,E1 -23396.001,E2 -23396.001} C_VEL
LIN {X 0,Y 163.277,Z 466.793,A -85,B 0,C 180,E1 -23399.383,E2 -23399.383} C_VEL
LIN {X 0,Y 163.315,Z 474.718,A -85,B 0,C 180,E1 -23402.466,E2 -23402.466} C_VEL
LIN {X 0,Y 164.026,Z 482.376,A -85,B 0,C 180,E1 -23406.149,E2 -23406.149} C_VEL
LIN {X 0,Y 165.552,Z 488.58,A -85,B 0,C 180,E1 -23409.777,E2 -23409.777} C_VEL
LIN {X 0,Y 168.023,Z 493.464,A -85,B 0,C 180,E1 -23413.3,E2 -23413.3} C_VEL
LIN {X 0,Y 171.26,Z 497.154,A -85,B 0,C 180,E1 -23416.694,E2 -23416.694} C_VEL
LIN {X 0,Y 173.879,Z 499.02,A -85,B 0,C 180,E1 -23418.866,E2 -23418.866} C_VEL
LIN {X 0,Y 176.85,Z 500.366,A -85,B 0,C 180,E1 -23420.957,E2 -23420.957} C_VEL
LIN {X 0,Y 180.093,Z 501.284,A -85,B 0,C 180,E1 -23422.97,E2 -23422.97} C_VEL
LIN {X 0,Y 183.59,Z 501.705,A -85,B 0,C 180,E1 -23424.903,E2 -23424.903} C_VEL
LIN {X 0,Y 187.375,Z 501.706,A -85,B 0,C 180,E1 -23426.75,E2 -23426.75} C_VEL
LIN {X 0,Y 193.56,Z 500.81,A -85,B 0,C 180,E1 -23429.375,E2 -23429.375} C_VEL
LIN {X 0,Y 195.65,Z 500.333,A -85,B 0,C 180,E1 -23430.192,E2 -23430.192} C_VEL
LIN {X 0,Y 199.494,Z 499.211,A -85,B 0,C 180,E1 -23431.9,E2 -23431.9} C_VEL
LIN {X 0,Y 201.841,Z 498.413,A -85,B 0,C 180,E1 -23433.856,E2 -23433.856} C_VEL
LIN {X 0,Y 203.9,Z 497.738,A -85,B 0,C 180,E1 -23435.87,E2 -23435.87} C_VEL
LIN {X 0,Y 205.506,Z 497.329,A -85,B 0,C 180,E1 -23438.133,E2 -23438.133} C_VEL
LIN {X 0,Y 206.462,Z 497.43,A -85,B 0,C 180,E1 -23440.298,E2 -23440.298} C_VEL
LIN {X 0,Y 207.061,Z 498.075,A -85,B 0,C 180,E1 -23442.753,E2 -23442.753} C_VEL
LIN {X 0,Y 207.219,Z 499.413,A -85,B 0,C 180,E1 -23445.417,E2 -23445.417} C_VEL
LIN {X 0,Y 206.758,Z 500.792,A -85,B 0,C 180,E1 -23447.169,E2 -23447.169} C_VEL
LIN {X 0,Y 202.999,Z 503.72,A -85,B 0,C 180,E1 -23448.867,E2 -23448.867} C_VEL
LIN {X 0,Y 196.256,Z 507.91,A -85,B 0,C 180,E1 -23451.194,E2 -23451.194} C_VEL
LIN {X 0,Y 189.674,Z 511.355,A -85,B 0,C 180,E1 -23453.64,E2 -23453.64} C_VEL
LIN {X 0,Y 185.542,Z 513.223,A -85,B 0,C 180,E1 -23455.377,E2 -23455.377} C_VEL
LIN {X 0,Y 178.458,Z 516,A -85,B 0,C 180,E1 -23459.205,E2 -23459.205} C_VEL
LIN {X 0,Y 172.627,Z 517.603,A -85,B 0,C 180,E1 -23463.395,E2 -23463.395} C_VEL
LIN {X 0,Y 168.262,Z 518,A -85,B 0,C 180,E1 -23467.919,E2 -23467.919} C_VEL
LIN {X 0,Y 165.388,Z 517.252,A -85,B 0,C 180,E1 -23472.695,E2 -23472.695} C_VEL
LIN {X 0,Y 164.137,Z 515.344,A -85,B 0,C 180,E1 -23477.637,E2 -23477.637} C_VEL
LIN {X 0,Y 164.495,Z 512.178,A -85,B 0,C 180,E1 -23482.635,E2 -23482.635} C_VEL
LIN {X 0,Y 165.958,Z 507.398,A -85,B 0,C 180,E1 -23487.572,E2 -23487.572} C_VEL
LIN {X 0,Y 166.329,Z 503.997,A -85,B 0,C 180,E1 -23490,E2 -23490} C_VEL
LIN {X 0,Y 166.324,Z 498.571,A -85,B 0,C 180,E1 -23493.027,E2 -23493.027} C_VEL
LIN {X 0,Y 166.011,Z 491.497,A -85,B 0,C 180,E1 -23496.075,E2 -23496.075} C_VEL
LIN {X 0,Y 166.023,Z 482.758,A -85,B 0,C 180,E1 -23499.134,E2 -23499.134} C_VEL
LIN {X 0,Y 166.325,Z 471.72,A -85,B 0,C 180,E1 -23502.197,E2 -23502.197} C_VEL
LIN {X 0,Y 166.478,Z 467.028,A -85,B 0,C 180,E1 -23503.277,E2 -23503.277} C_VEL
LIN {X 0,Y 165.105,Z 455.019,A -85,B 0,C 180,E1 -23505.429,E2 -23505.429} C_VEL
LIN {X 0,Y 164.303,Z 441.693,A -85,B 0,C 180,E1 -23507.262,E2 -23507.262} C_VEL
LIN {X 0,Y 164.25,Z 433.791,A -85,B 0,C 180,E1 -23508.163,E2 -23508.163} C_VEL
LIN {X 0,Y 165.896,Z 423.197,A -85,B 0,C 180,E1 -23516.649,E2 -23516.649} C_VEL
LIN {X 0,Y 165.835,Z 420.815,A -85,B 0,C 180,E1 -23518.519,E2 -23518.519} C_VEL
LIN {X 0,Y 164.713,Z 418.447,A -85,B 0,C 180,E1 -23520.376,E2 -23520.376} C_VEL
LIN {X 0,Y 160.282,Z 412.253,A -85,B 0,C 180,E1 -23525.44,E2 -23525.44} C_VEL
LIN {X 0,Y 159.647,Z 410.68,A -85,B 0,C 180,E1 -23526.769,E2 -23526.769} C_VEL
LIN {X 0,Y 158.262,Z 404.862,A -85,B 0,C 180,E1 -23531.767,E2 -23531.767} C_VEL
LIN {X 0,Y 157.431,Z 400.871,A -85,B 0,C 180,E1 -23535.457,E2 -23535.457} C_VEL
LIN {X 0,Y 157.239,Z 400.898,A -85,B 0,C 180,E1 -23541.263,E2 -23541.263} C_VEL
LIN {X 0,Y 157.29,Z 400.888,A -85,B 0,C 180,E1 -23544.489,E2 -23544.489} C_VEL
LIN {X 0,Y 157.294,Z 400.891,A -85,B 0,C 180,E1 -23548.095,E2 -23548.095} C_VEL
LIN {X 0,Y 157.322,Z 400.885,A -85,B 0,C 180,E1 -23553.466,E2 -23553.466} C_VEL
LIN {X 0,Y 157.394,Z 400.88,A -85,B 0,C 180,E1 -23559.667,E2 -23559.667} C_VEL
LIN {X 0,Y 157.479,Z 400.866,A -85,B 0,C 180,E1 -23564.468,E2 -23564.468} C_VEL
LIN {X 0,Y 157.773,Z 400.829,A -85,B 0,C 180,E1 -23569.736,E2 -23569.736} C_VEL
LIN {X 0,Y 157.825,Z 400.822,A -85,B 0,C 180,E1 -23572.323,E2 -23572.323} C_VEL
LIN {X 0,Y 158.259,Z 400.766,A -85,B 0,C 180,E1 -23580,E2 -23580} C_VEL
LIN {X 0,Y 157.825,Z 400.82,A -85,B 0,C 180,E1 -23587.677,E2 -23587.677} C_VEL
LIN {X 0,Y 157.706,Z 400.84,A -85,B 0,C 180,E1 -23591.363,E2 -23591.363} C_VEL
LIN {X 0,Y 157.486,Z 400.864,A -85,B 0,C 180,E1 -23595.531,E2 -23595.531} C_VEL
LIN {X 0,Y 157.372,Z 400.882,A -85,B 0,C 180,E1 -23600.933,E2 -23600.933} C_VEL
LIN {X 0,Y 157.315,Z 400.884,A -85,B 0,C 180,E1 -23606.685,E2 -23606.685} C_VEL
LIN {X 0,Y 157.281,Z 400.892,A -85,B 0,C 180,E1 -23612.426,E2 -23612.426} C_VEL
LIN {X 0,Y 157.268,Z 400.892,A -85,B 0,C 180,E1 -23616.45,E2 -23616.45} C_VEL
LIN {X 0,Y 157.211,Z 400.898,A -85,B 0,C 180,E1 -23622.111,E2 -23622.111} C_VEL
LIN {X 0,Y 157.213,Z 400.901,A -85,B 0,C 180,E1 -23627.891,E2 -23627.891} C_VEL
LIN {X 0,Y 157.284,Z 400.891,A -85,B 0,C 180,E1 -23633.544,E2 -23633.544} C_VEL
LIN {X 0,Y 157.296,Z 400.89,A -85,B 0,C 180,E1 -23638.095,E2 -23638.095} C_VEL
LIN {X 0,Y 157.324,Z 400.887,A -85,B 0,C 180,E1 -23643.467,E2 -23643.467} C_VEL
LIN {X 0,Y 157.448,Z 400.868,A -85,B 0,C 180,E1 -23649.616,E2 -23649.616} C_VEL
LIN {X 0,Y 157.49,Z 400.866,A -85,B 0,C 180,E1 -23654.47,E2 -23654.47} C_VEL
LIN {X 0,Y 157.736,Z 400.835,A -85,B 0,C 180,E1 -23659.734,E2 -23659.734} C_VEL
LIN {X 0,Y 157.811,Z 400.827,A -85,B 0,C 180,E1 -23662.323,E2 -23662.323} C_VEL
LIN {X 0,Y 158.261,Z 400.773,A -85,B 0,C 180,E1 -23670,E2 -23670} C_VEL
LIN {X 0,Y 157.77,Z 400.832,A -85,B 0,C 180,E1 -23677.68,E2 -23677.68} C_VEL
LIN {X 0,Y 157.64,Z 400.846,A -85,B 0,C 180,E1 -23681.239,E2 -23681.239} C_VEL
LIN {X 0,Y 157.464,Z 400.869,A -85,B 0,C 180,E1 -23685.534,E2 -23685.534} C_VEL
LIN {X 0,Y 157.374,Z 400.877,A -85,B 0,C 180,E1 -23690.933,E2 -23690.933} C_VEL
LIN {X 0,Y 157.317,Z 400.888,A -85,B 0,C 180,E1 -23696.686,E2 -23696.686} C_VEL
LIN {X 0,Y 157.281,Z 400.891,A -85,B 0,C 180,E1 -23702.427,E2 -23702.427} C_VEL
LIN {X 0,Y 157.285,Z 400.89,A -85,B 0,C 180,E1 -23706.457,E2 -23706.457} C_VEL
LIN {X 0,Y 157.215,Z 400.901,A -85,B 0,C 180,E1 -23712.11,E2 -23712.11} C_VEL
LIN {X 0,Y 157.215,Z 400.897,A -85,B 0,C 180,E1 -23717.89,E2 -23717.89} C_VEL
LIN {X 0,Y 157.35,Z 400.882,A -85,B 0,C 180,E1 -23723.512,E2 -23723.512} C_VEL
LIN {X 0,Y 157.69,Z 400.839,A -85,B 0,C 180,E1 -23728.589,E2 -23728.589} C_VEL
LIN {X 0,Y 157.557,Z 401.016,A -85,B 0,C 180,E1 -23729.249,E2 -23729.249} C_VEL
LIN {X 0,Y 156.685,Z 406.269,A -85,B 0,C 180,E1 -23734.911,E2 -23734.911} C_VEL
LIN {X 0,Y 155.982,Z 412.083,A -85,B 0,C 180,E1 -23741.12,E2 -23741.12} C_VEL
LIN {X 0,Y 156.163,Z 420.062,A -85,B 0,C 180,E1 -23749.465,E2 -23749.465} C_VEL
LIN {X 0,Y 157.552,Z 433.504,A -85,B 0,C 180,E1 -23751.47,E2 -23751.47} C_VEL
LIN {X 0,Y 157.148,Z 445.315,A -85,B 0,C 180,E1 -23753.903,E2 -23753.903} C_VEL
LIN {X 0,Y 156.798,Z 456.394,A -85,B 0,C 180,E1 -23756.788,E2 -23756.788} C_VEL
LIN {X 0,Y 156.378,Z 466.16,A -85,B 0,C 180,E1 -23760,E2 -23760} C_VEL
LIN {X 0,Y 156.588,Z 475.591,A -85,B 0,C 180,E1 -23763.86,E2 -23763.86} C_VEL
LIN {X 0,Y 157.503,Z 483.255,A -85,B 0,C 180,E1 -23767.693,E2 -23767.693} C_VEL
LIN {X 0,Y 159.37,Z 489.353,A -85,B 0,C 180,E1 -23771.446,E2 -23771.446} C_VEL
LIN {X 0,Y 162.15,Z 494.282,A -85,B 0,C 180,E1 -23775.073,E2 -23775.073} C_VEL
LIN {X 0,Y 165.776,Z 497.981,A -85,B 0,C 180,E1 -23778.54,E2 -23778.54} C_VEL
LIN {X 0,Y 170.224,Z 500.633,A -85,B 0,C 180,E1 -23781.813,E2 -23781.813} C_VEL
LIN {X 0,Y 173.579,Z 501.82,A -85,B 0,C 180,E1 -23783.884,E2 -23783.884} C_VEL
LIN {X 0,Y 177.205,Z 502.538,A -85,B 0,C 180,E1 -23785.866,E2 -23785.866} C_VEL
LIN {X 0,Y 181.102,Z 502.825,A -85,B 0,C 180,E1 -23787.755,E2 -23787.755} C_VEL
LIN {X 0,Y 187.339,Z 502.417,A -85,B 0,C 180,E1 -23790.362,E2 -23790.362} C_VEL
LIN {X 0,Y 189.657,Z 502.072,A -85,B 0,C 180,E1 -23791.251,E2 -23791.251} C_VEL
LIN {X 0,Y 193.66,Z 501.221,A -85,B 0,C 180,E1 -23792.981,E2 -23792.981} C_VEL
LIN {X 0,Y 196.065,Z 500.745,A -85,B 0,C 180,E1 -23794.996,E2 -23794.996} C_VEL
LIN {X 0,Y 198.096,Z 500.364,A -85,B 0,C 180,E1 -23797.094,E2 -23797.094} C_VEL
LIN {X 0,Y 199.535,Z 500.376,A -85,B 0,C 180,E1 -23799.345,E2 -23799.345} C_VEL
LIN {X 0,Y 200.466,Z 500.78,A -85,B 0,C 180,E1 -23801.768,E2 -23801.768} C_VEL
LIN {X 0,Y 200.755,Z 501.865,A -85,B 0,C 180,E1 -23804.44,E2 -23804.44} C_VEL
LIN {X 0,Y 200.665,Z 502.522,A -85,B 0,C 180,E1 -23805.534,E2 -23805.534} C_VEL
LIN {X 0,Y 199.765,Z 503.583,A -85,B 0,C 180,E1 -23806.682,E2 -23806.682} C_VEL
LIN {X 0,Y 195.536,Z 506.171,A -85,B 0,C 180,E1 -23808.322,E2 -23808.322} C_VEL
LIN {X 0,Y 188.461,Z 509.7,A -85,B 0,C 180,E1 -23810.657,E2 -23810.657} C_VEL
LIN {X 0,Y 179.76,Z 513.229,A -85,B 0,C 180,E1 -23814.094,E2 -23814.094} C_VEL
LIN {X 0,Y 172.411,Z 515.527,A -85,B 0,C 180,E1 -23817.999,E2 -23817.999} C_VEL
LIN {X 0,Y 166.348,Z 516.678,A -85,B 0,C 180,E1 -23822.306,E2 -23822.306} C_VEL
LIN {X 0,Y 161.771,Z 516.688,A -85,B 0,C 180,E1 -23826.983,E2 -23826.983} C_VEL
LIN {X 0,Y 158.766,Z 515.552,A -85,B 0,C 180,E1 -23831.948,E2 -23831.948} C_VEL
LIN {X 0,Y 157.457,Z 513.333,A -85,B 0,C 180,E1 -23837.104,E2 -23837.104} C_VEL
LIN {X 0,Y 157.827,Z 509.8,A -85,B 0,C 180,E1 -23842.322,E2 -23842.322} C_VEL
LIN {X 0,Y 158.869,Z 506.192,A -85,B 0,C 180,E1 -23846.195,E2 -23846.195} C_VEL
LIN {X 0,Y 159.655,Z 503.005,A -85,B 0,C 180,E1 -23848.738,E2 -23848.738} C_VEL
LIN {X 0,Y 159.736,Z 497.69,A -85,B 0,C 180,E1 -23851.891,E2 -23851.891} C_VEL
LIN {X 0,Y 159.375,Z 490.777,A -85,B 0,C 180,E1 -23855.059,E2 -23855.059} C_VEL
LIN {X 0,Y 159.275,Z 482.229,A -85,B 0,C 180,E1 -23858.245,E2 -23858.245} C_VEL
LIN {X 0,Y 159.47,Z 471.371,A -85,B 0,C 180,E1 -23861.438,E2 -23861.438} C_VEL
LIN {X 0,Y 159.576,Z 466.02,A -85,B 0,C 180,E1 -23862.721,E2 -23862.721} C_VEL
LIN {X 0,Y 158.123,Z 453.945,A -85,B 0,C 180,E1 -23864.957,E2 -23864.957} C_VEL
LIN {X 0,Y 157.386,Z 441.836,A -85,B 0,C 180,E1 -23866.706,E2 -23866.706} C_VEL
LIN {X 0,Y 157.281,Z 433.446,A -85,B 0,C 180,E1 -23867.722,E2 -23867.722} C_VEL
LIN {X 0,Y 160.248,Z 418.563,A -85,B 0,C 180,E1 -23880.288,E2 -23880.288} C_VEL
LIN {X 0,Y 160.841,Z 416.915,A -85,B 0,C 180,E1 -23881.624,E2 -23881.624} C_VEL
LIN {X 0,Y 160.92,Z 415.657,A -85,B 0,C 180,E1 -23882.644,E2 -23882.644} C_VEL
LIN {X 0,Y 159.647,Z 410.68,A -85,B 0,C 180,E1 -23886.769,E2 -23886.769} C_VEL
LIN {X 0,Y 158.598,Z 409.233,A -85,B 0,C 180,E1 -23888.039,E2 -23888.039} C_VEL
LIN {X 0,Y 155.231,Z 407.13,A -85,B 0,C 180,E1 -23890.014,E2 -23890.014} C_VEL
LIN {X 0,Y 151.838,Z 405.065,A -85,B 0,C 180,E1 -23892.07,E2 -23892.07} C_VEL
LIN {X 0,Y 150.801,Z 403.642,A -85,B 0,C 180,E1 -23893.438,E2 -23893.438} C_VEL
LIN {X 0,Y 150.392,Z 401.748,A -85,B 0,C 180,E1 -23895.22,E2 -23895.22} C_VEL
LIN {X 0,Y 150.211,Z 401.773,A -85,B 0,C 180,E1 -23902.538,E2 -23902.538} C_VEL
LIN {X 0,Y 150.218,Z 401.769,A -85,B 0,C 180,E1 -23907.366,E2 -23907.366} C_VEL
LIN {X 0,Y 150.244,Z 401.766,A -85,B 0,C 180,E1 -23912.718,E2 -23912.718} C_VEL
LIN {X 0,Y 150.351,Z 401.756,A -85,B 0,C 180,E1 -23919.207,E2 -23919.207} C_VEL
LIN {X 0,Y 150.383,Z 401.748,A -85,B 0,C 180,E1 -23923.716,E2 -23923.716} C_VEL
LIN {X 0,Y 150.69,Z 401.714,A -85,B 0,C 180,E1 -23929.248,E2 -23929.248} C_VEL
LIN {X 0,Y 150.764,Z 401.701,A -85,B 0,C 180,E1 -23931.961,E2 -23931.961} C_VEL
LIN {X 0,Y 151.219,Z 401.643,A -85,B 0,C 180,E1 -23940,E2 -23940} C_VEL
LIN {X 0,Y 150.764,Z 401.699,A -85,B 0,C 180,E1 -23948.039,E2 -23948.039} C_VEL
LIN {X 0,Y 150.635,Z 401.722,A -85,B 0,C 180,E1 -23951.546,E2 -23951.546} C_VEL
LIN {X 0,Y 150.391,Z 401.747,A -85,B 0,C 180,E1 -23956.284,E2 -23956.284} C_VEL
LIN {X 0,Y 150.352,Z 401.756,A -85,B 0,C 180,E1 -23960.794,E2 -23960.794} C_VEL
LIN {X 0,Y 150.246,Z 401.768,A -85,B 0,C 180,E1 -23967.283,E2 -23967.283} C_VEL
LIN {X 0,Y 150.22,Z 401.771,A -85,B 0,C 180,E1 -23972.636,E2 -23972.636} C_VEL
LIN {X 0,Y 150.177,Z 401.778,A -85,B 0,C 180,E1 -23977.472,E2 -23977.472} C_VEL
LIN {X 0,Y 150.15,Z 401.777,A -85,B 0,C 180,E1 -23981.505,E2 -23981.505} C_VEL
LIN {X 0,Y 150.126,Z 401.783,A -85,B 0,C 180,E1 -23985.396,E2 -23985.396} C_VEL
LIN {X 0,Y 150.157,Z 401.779,A -85,B 0,C 180,E1 -23989.061,E2 -23989.061} C_VEL
LIN {X 0,Y 150.216,Z 401.77,A -85,B 0,C 180,E1 -23992.69,E2 -23992.69} C_VEL
LIN {X 0,Y 150.219,Z 401.771,A -85,B 0,C 180,E1 -23997.366,E2 -23997.366} C_VEL
LIN {X 0,Y 150.246,Z 401.77,A -85,B 0,C 180,E1 -24002.718,E2 -24002.718} C_VEL
LIN {X 0,Y 150.391,Z 401.746,A -85,B 0,C 180,E1 -24009.169,E2 -24009.169} C_VEL
LIN {X 0,Y 150.399,Z 401.75,A -85,B 0,C 180,E1 -24013.718,E2 -24013.718} C_VEL
LIN {X 0,Y 150.66,Z 401.715,A -85,B 0,C 180,E1 -24019.247,E2 -24019.247} C_VEL
LIN {X 0,Y 150.747,Z 401.708,A -85,B 0,C 180,E1 -24021.961,E2 -24021.961} C_VEL
LIN {X 0,Y 151.222,Z 401.65,A -85,B 0,C 180,E1 -24030.001,E2 -24030.001} C_VEL
LIN {X 0,Y 150.707,Z 401.713,A -85,B 0,C 180,E1 -24038.043,E2 -24038.043} C_VEL
LIN {X 0,Y 150.58,Z 401.726,A -85,B 0,C 180,E1 -24041.439,E2 -24041.439} C_VEL
LIN {X 0,Y 150.372,Z 401.753,A -85,B 0,C 180,E1 -24046.286,E2 -24046.286} C_VEL
LIN {X 0,Y 150.354,Z 401.751,A -85,B 0,C 180,E1 -24050.794,E2 -24050.794} C_VEL
LIN {X 0,Y 150.247,Z 401.77,A -85,B 0,C 180,E1 -24057.283,E2 -24057.283} C_VEL
LIN {X 0,Y 150.221,Z 401.771,A -85,B 0,C 180,E1 -24062.635,E2 -24062.635} C_VEL
LIN {X 0,Y 150.214,Z 401.769,A -85,B 0,C 180,E1 -24067.462,E2 -24067.462} C_VEL
LIN {X 0,Y 150.157,Z 401.781,A -85,B 0,C 180,E1 -24071.507,E2 -24071.507} C_VEL
LIN {X 0,Y 150.128,Z 401.781,A -85,B 0,C 180,E1 -24075.396,E2 -24075.396} C_VEL
LIN {X 0,Y 150.158,Z 401.778,A -85,B 0,C 180,E1 -24079.061,E2 -24079.061} C_VEL
LIN {X 0,Y 150.241,Z 401.77,A -85,B 0,C 180,E1 -24082.678,E2 -24082.678} C_VEL
LIN {X 0,Y 150.508,Z 401.726,A -85,B 0,C 180,E1 -24087.195,E2 -24087.195} C_VEL
LIN {X 0,Y 150.436,Z 401.803,A -85,B 0,C 180,E1 -24089.466,E2 -24089.466} C_VEL
LIN {X 0,Y 149.58,Z 406.725,A -85,B 0,C 180,E1 -24094.984,E2 -24094.984} C_VEL
LIN {X 0,Y 148.922,Z 411.876,A -85,B 0,C 180,E1 -24100.71,E2 -24100.71} C_VEL
LIN {X 0,Y 149.252,Z 420.443,A -85,B 0,C 180,E1 -24110.061,E2 -24110.061} C_VEL
LIN {X 0,Y 150.605,Z 432.853,A -85,B 0,C 180,E1 -24111.952,E2 -24111.952} C_VEL
LIN {X 0,Y 150.24,Z 444.039,A -85,B 0,C 180,E1 -24114.295,E2 -24114.295} C_VEL
LIN {X 0,Y 149.961,Z 454.255,A -85,B 0,C 180,E1 -24116.978,E2 -24116.978} C_VEL
LIN {X 0,Y 149.539,Z 465.251,A -85,B 0,C 180,E1 -24120.673,E2 -24120.673} C_VEL
LIN {X 0,Y 149.697,Z 473.526,A -85,B 0,C 180,E1 -24124.038,E2 -24124.038} C_VEL
LIN {X 0,Y 150.603,Z 481.603,A -85,B 0,C 180,E1 -24128.048,E2 -24128.048} C_VEL
LIN {X 0,Y 152.502,Z 488.191,A -85,B 0,C 180,E1 -24131.969,E2 -24131.969} C_VEL
LIN {X 0,Y 155.342,Z 493.513,A -85,B 0,C 180,E1 -24135.751,E2 -24135.751} C_VEL
LIN {X 0,Y 159.052,Z 497.629,A -85,B 0,C 180,E1 -24139.354,E2 -24139.354} C_VEL
LIN {X 0,Y 163.634,Z 500.701,A -85,B 0,C 180,E1 -24142.74,E2 -24142.74} C_VEL
LIN {X 0,Y 167.117,Z 502.161,A -85,B 0,C 180,E1 -24144.869,E2 -24144.869} C_VEL
LIN {X 0,Y 170.854,Z 503.18,A -85,B 0,C 180,E1 -24146.903,E2 -24146.903} C_VEL
LIN {X 0,Y 174.883,Z 503.755,A -85,B 0,C 180,E1 -24148.832,E2 -24148.832} C_VEL
LIN {X 0,Y 181.308,Z 503.796,A -85,B 0,C 180,E1 -24151.484,E2 -24151.484} C_VEL
LIN {X 0,Y 183.706,Z 503.604,A -85,B 0,C 180,E1 -24152.384,E2 -24152.384} C_VEL
LIN {X 0,Y 187.828,Z 503.066,A -85,B 0,C 180,E1 -24154.143,E2 -24154.143} C_VEL
LIN {X 0,Y 190.244,Z 502.879,A -85,B 0,C 180,E1 -24156.233,E2 -24156.233} C_VEL
LIN {X 0,Y 192.183,Z 502.858,A -85,B 0,C 180,E1 -24158.439,E2 -24158.439} C_VEL
LIN {X 0,Y 193.436,Z 503.194,A -85,B 0,C 180,E1 -24160.843,E2 -24160.843} C_VEL
LIN {X 0,Y 194.088,Z 504.12,A -85,B 0,C 180,E1 -24163.596,E2 -24163.596} C_VEL
LIN {X 0,Y 192.613,Z 505.865,A -85,B 0,C 180,E1 -24166.11,E2 -24166.11} C_VEL
LIN {X 0,Y 187.891,Z 508.105,A -85,B 0,C 180,E1 -24167.678,E2 -24167.678} C_VEL
LIN {X 0,Y 178.46,Z 511.743,A -85,B 0,C 180,E1 -24170.942,E2 -24170.942} C_VEL
LIN {X 0,Y 174.078,Z 513.077,A -85,B 0,C 180,E1 -24172.728,E2 -24172.728} C_VEL
LIN {X 0,Y 166.454,Z 514.881,A -85,B 0,C 180,E1 -24176.709,E2 -24176.709} C_VEL
LIN {X 0,Y 160.145,Z 515.579,A -85,B 0,C 180,E1 -24181.135,E2 -24181.135} C_VEL
LIN {X 0,Y 155.362,Z 515.194,A -85,B 0,C 180,E1 -24185.975,E2 -24185.975} C_VEL
LIN {X 0,Y 152.217,Z 513.725,A -85,B 0,C 180,E1 -24191.143,E2 -24191.143} C_VEL
LIN {X 0,Y 150.853,Z 511.098,A -85,B 0,C 180,E1 -24196.529,E2 -24196.529} C_VEL
LIN {X 0,Y 151.236,Z 507.303,A -85,B 0,C 180,E1 -24201.986,E2 -24201.986} C_VEL
LIN {X 0,Y 152.371,Z 503.381,A -85,B 0,C 180,E1 -24206.032,E2 -24206.032} C_VEL
LIN {X 0,Y 152.869,Z 501.831,A -85,B 0,C 180,E1 -24207.364,E2 -24207.364} C_VEL
LIN {X 0,Y 153.172,Z 497.968,A -85,B 0,C 180,E1 -24209.999,E2 -24209.999} C_VEL
LIN {X 0,Y 152.977,Z 492.909,A -85,B 0,C 180,E1 -24212.633,E2 -24212.633} C_VEL
LIN {X 0,Y 152.693,Z 485.119,A -85,B 0,C 180,E1 -24215.944,E2 -24215.944} C_VEL
LIN {X 0,Y 152.555,Z 475.269,A -85,B 0,C 180,E1 -24219.278,E2 -24219.278} C_VEL
LIN {X 0,Y 152.8,Z 465.493,A -85,B 0,C 180,E1 -24221.945,E2 -24221.945} C_VEL
LIN {X 0,Y 151.328,Z 453.799,A -85,B 0,C 180,E1 -24224.231,E2 -24224.231} C_VEL
LIN {X 0,Y 150.43,Z 440.273,A -85,B 0,C 180,E1 -24226.279,E2 -24226.279} C_VEL
LIN {X 0,Y 150.33,Z 433.171,A -85,B 0,C 180,E1 -24227.164,E2 -24227.164} C_VEL
LIN {X 0,Y 150.626,Z 426.287,A -85,B 0,C 180,E1 -24233.365,E2 -24233.365} C_VEL
LIN {X 0,Y 153.099,Z 418.429,A -85,B 0,C 180,E1 -24240.328,E2 -24240.328} C_VEL
LIN {X 0,Y 153.715,Z 416.81,A -85,B 0,C 180,E1 -24241.721,E2 -24241.721} C_VEL
LIN {X 0,Y 153.297,Z 413.715,A -85,B 0,C 180,E1 -24244.389,E2 -24244.389} C_VEL
LIN {X 0,Y 151.489,Z 406.842,A -85,B 0,C 180,E1 -24250.503,E2 -24250.503} C_VEL
LIN {X 0,Y 150.801,Z 403.642,A -85,B 0,C 180,E1 -24253.438,E2 -24253.438} C_VEL
LIN {X 0,Y 150.153,Z 402.566,A -85,B 0,C 180,E1 -24254.836,E2 -24254.836} C_VEL
LIN {X 0,Y 148.498,Z 402.059,A -85,B 0,C 180,E1 -24256.992,E2 -24256.992} C_VEL
LIN {X 0,Y 144.113,Z 402.537,A -85,B 0,C 180,E1 -24262.238,E2 -24262.238} C_VEL
LIN {X 0,Y 143.106,Z 402.651,A -85,B 0,C 180,E1 -24265.44,E2 -24265.44} C_VEL
LIN {X 0,Y 143.185,Z 402.645,A -85,B 0,C 180,E1 -24267.322,E2 -24267.322} C_VEL
LIN {X 0,Y 143.19,Z 402.647,A -85,B 0,C 180,E1 -24272.063,E2 -24272.063} C_VEL
LIN {X 0,Y 143.277,Z 402.637,A -85,B 0,C 180,E1 -24278.745,E2 -24278.745} C_VEL
LIN {X 0,Y 143.317,Z 402.625,A -85,B 0,C 180,E1 -24282.889,E2 -24282.889} C_VEL
LIN {X 0,Y 143.603,Z 402.595,A -85,B 0,C 180,E1 -24288.711,E2 -24288.711} C_VEL
LIN {X 0,Y 143.685,Z 402.581,A -85,B 0,C 180,E1 -24291.562,E2 -24291.562} C_VEL
LIN {X 0,Y 144.178,Z 402.52,A -85,B 0,C 180,E1 -24300,E2 -24300} C_VEL
LIN {X 0,Y 143.685,Z 402.58,A -85,B 0,C 180,E1 -24308.438,E2 -24308.438} C_VEL
LIN {X 0,Y 143.571,Z 402.601,A -85,B 0,C 180,E1 -24311.758,E2 -24311.758} C_VEL
LIN {X 0,Y 143.323,Z 402.627,A -85,B 0,C 180,E1 -24317.111,E2 -24317.111} C_VEL
LIN {X 0,Y 143.278,Z 402.639,A -85,B 0,C 180,E1 -24321.256,E2 -24321.256} C_VEL
LIN {X 0,Y 143.193,Z 402.646,A -85,B 0,C 180,E1 -24327.939,E2 -24327.939} C_VEL
LIN {X 0,Y 143.147,Z 402.648,A -85,B 0,C 180,E1 -24333.423,E2 -24333.423} C_VEL
LIN {X 0,Y 143.062,Z 402.663,A -85,B 0,C 180,E1 -24339.69,E2 -24339.69} C_VEL
LIN {X 0,Y 143.056,Z 402.661,A -85,B 0,C 180,E1 -24343.456,E2 -24343.456} C_VEL
LIN {X 0,Y 143.068,Z 402.663,A -85,B 0,C 180,E1 -24347.464,E2 -24347.464} C_VEL
LIN {X 0,Y 143.107,Z 402.652,A -85,B 0,C 180,E1 -24351.791,E2 -24351.791} C_VEL
LIN {X 0,Y 143.187,Z 402.647,A -85,B 0,C 180,E1 -24357.323,E2 -24357.323} C_VEL
LIN {X 0,Y 143.163,Z 402.651,A -85,B 0,C 180,E1 -24363.781,E2 -24363.781} C_VEL
LIN {X 0,Y 143.345,Z 402.625,A -85,B 0,C 180,E1 -24369.929,E2 -24369.929} C_VEL
LIN {X 0,Y 143.385,Z 402.622,A -85,B 0,C 180,E1 -24375.814,E2 -24375.814} C_VEL
LIN {X 0,Y 143.596,Z 402.596,A -85,B 0,C 180,E1 -24378.711,E2 -24378.711} C_VEL
LIN {X 0,Y 143.667,Z 402.589,A -85,B 0,C 180,E1 -24381.562,E2 -24381.562} C_VEL
LIN {X 0,Y 144.18,Z 402.527,A -85,B 0,C 180,E1 -24390.001,E2 -24390.001} C_VEL
LIN {X 0,Y 143.629,Z 402.594,A -85,B 0,C 180,E1 -24398.442,E2 -24398.442} C_VEL
LIN {X 0,Y 143.508,Z 402.605,A -85,B 0,C 180,E1 -24401.632,E2 -24401.632} C_VEL
LIN {X 0,Y 143.31,Z 402.633,A -85,B 0,C 180,E1 -24407.113,E2 -24407.113} C_VEL
LIN {X 0,Y 143.28,Z 402.632,A -85,B 0,C 180,E1 -24411.256,E2 -24411.256} C_VEL
LIN {X 0,Y 143.193,Z 402.645,A -85,B 0,C 180,E1 -24417.938,E2 -24417.938} C_VEL
LIN {X 0,Y 143.171,Z 402.651,A -85,B 0,C 180,E1 -24423.436,E2 -24423.436} C_VEL
LIN {X 0,Y 143.077,Z 402.659,A -85,B 0,C 180,E1 -24429.686,E2 -24429.686} C_VEL
LIN {X 0,Y 143.059,Z 402.665,A -85,B 0,C 180,E1 -24433.455,E2 -24433.455} C_VEL
LIN {X 0,Y 143.069,Z 402.659,A -85,B 0,C 180,E1 -24437.464,E2 -24437.464} C_VEL
LIN {X 0,Y 143.216,Z 402.642,A -85,B 0,C 180,E1 -24443.923,E2 -24443.923} C_VEL
LIN {X 0,Y 143.461,Z 402.603,A -85,B 0,C 180,E1 -24447.393,E2 -24447.393} C_VEL
LIN {X 0,Y 143.271,Z 402.67,A -85,B 0,C 180,E1 -24449.814,E2 -24449.814} C_VEL
LIN {X 0,Y 142.439,Z 407.29,A -85,B 0,C 180,E1 -24455.204,E2 -24455.204} C_VEL
LIN {X 0,Y 141.749,Z 412.678,A -85,B 0,C 180,E1 -24461.47,E2 -24461.47} C_VEL
LIN {X 0,Y 141.943,Z 419.93,A -85,B 0,C 180,E1 -24469.787,E2 -24469.787} C_VEL
LIN {X 0,Y 142.349,Z 420.747,A -85,B 0,C 180,E1 -24470.696,E2 -24470.696} C_VEL
LIN {X 0,Y 143.68,Z 432.855,A -85,B 0,C 180,E1 -24472.623,E2 -24472.623} C_VEL
LIN {X 0,Y 143.345,Z 443.904,A -85,B 0,C 180,E1 -24475.078,E2 -24475.078} C_VEL
LIN {X 0,Y 143.091,Z 454.076,A -85,B 0,C 180,E1 -24477.889,E2 -24477.889} C_VEL
LIN {X 0,Y 142.736,Z 464.32,A -85,B 0,C 180,E1 -24481.411,E2 -24481.411} C_VEL
LIN {X 0,Y 142.974,Z 472.689,A -85,B 0,C 180,E1 -24484.935,E2 -24484.935} C_VEL
LIN {X 0,Y 144.01,Z 481.007,A -85,B 0,C 180,E1 -24489.126,E2 -24489.126} C_VEL
LIN {X 0,Y 146.069,Z 487.851,A -85,B 0,C 180,E1 -24493.211,E2 -24493.211} C_VEL
LIN {X 0,Y 149.743,Z 494.177,A -85,B 0,C 180,E1 -24497.762,E2 -24497.762} C_VEL
LIN {X 0,Y 153.897,Z 498.36,A -85,B 0,C 180,E1 -24501.428,E2 -24501.428} C_VEL
LIN {X 0,Y 157.089,Z 500.556,A -85,B 0,C 180,E1 -24503.744,E2 -24503.744} C_VEL
LIN {X 0,Y 160.692,Z 502.307,A -85,B 0,C 180,E1 -24505.936,E2 -24505.936} C_VEL
LIN {X 0,Y 164.54,Z 503.615,A -85,B 0,C 180,E1 -24508.024,E2 -24508.024} C_VEL
LIN {X 0,Y 168.711,Z 504.485,A -85,B 0,C 180,E1 -24509.992,E2 -24509.992} C_VEL
LIN {X 0,Y 175.531,Z 504.971,A -85,B 0,C 180,E1 -24512.773,E2 -24512.773} C_VEL
LIN {X 0,Y 177.806,Z 504.945,A -85,B 0,C 180,E1 -24513.598,E2 -24513.598} C_VEL
LIN {X 0,Y 181.996,Z 504.72,A -85,B 0,C 180,E1 -24515.397,E2 -24515.397} C_VEL
LIN {X 0,Y 184.336,Z 504.833,A -85,B 0,C 180,E1 -24517.591,E2 -24517.591} C_VEL
LIN {X 0,Y 186.155,Z 505.148,A -85,B 0,C 180,E1 -24519.927,E2 -24519.927} C_VEL
LIN {X 0,Y 186.715,Z 505.413,A -85,B 0,C 180,E1 -24521.165,E2 -24521.165} C_VEL
LIN {X 0,Y 187.045,Z 505.881,A -85,B 0,C 180,E1 -24522.558,E2 -24522.558} C_VEL
LIN {X 0,Y 186.66,Z 506.75,A -85,B 0,C 180,E1 -24524.325,E2 -24524.325} C_VEL
LIN {X 0,Y 182.712,Z 508.582,A -85,B 0,C 180,E1 -24526.182,E2 -24526.182} C_VEL
LIN {X 0,Y 173.023,Z 511.654,A -85,B 0,C 180,E1 -24529.465,E2 -24529.465} C_VEL
LIN {X 0,Y 168.506,Z 512.724,A -85,B 0,C 180,E1 -24531.272,E2 -24531.272} C_VEL
LIN {X 0,Y 160.61,Z 514.046,A -85,B 0,C 180,E1 -24535.329,E2 -24535.329} C_VEL
LIN {X 0,Y 154.051,Z 514.298,A -85,B 0,C 180,E1 -24539.878,E2 -24539.878} C_VEL
LIN {X 0,Y 149.056,Z 513.541,A -85,B 0,C 180,E1 -24544.89,E2 -24544.89} C_VEL
LIN {X 0,Y 145.762,Z 511.666,A -85,B 0,C 180,E1 -24550.274,E2 -24550.274} C_VEL
LIN {X 0,Y 144.318,Z 508.728,A -85,B 0,C 180,E1 -24555.907,E2 -24555.907} C_VEL
LIN {X 0,Y 144.724,Z 504.603,A -85,B 0,C 180,E1 -24561.623,E2 -24561.623} C_VEL
LIN {X 0,Y 145.953,Z 500.423,A -85,B 0,C 180,E1 -24565.857,E2 -24565.857} C_VEL
LIN {X 0,Y 146.431,Z 498.737,A -85,B 0,C 180,E1 -24567.248,E2 -24567.248} C_VEL
LIN {X 0,Y 146.666,Z 494.528,A -85,B 0,C 180,E1 -24569.999,E2 -24569.999} C_VEL
LIN {X 0,Y 146.326,Z 489.073,A -85,B 0,C 180,E1 -24572.752,E2 -24572.752} C_VEL
LIN {X 0,Y 146.016,Z 480.698,A -85,B 0,C 180,E1 -24576.217,E2 -24576.217} C_VEL
LIN {X 0,Y 145.97,Z 469.971,A -85,B 0,C 180,E1 -24579.701,E2 -24579.701} C_VEL
LIN {X 0,Y 146.097,Z 464.827,A -85,B 0,C 180,E1 -24581.094,E2 -24581.094} C_VEL
LIN {X 0,Y 144.529,Z 453.256,A -85,B 0,C 180,E1 -24583.457,E2 -24583.457} C_VEL
LIN {X 0,Y 143.623,Z 440.994,A -85,B 0,C 180,E1 -24585.43,E2 -24585.43} C_VEL
LIN {X 0,Y 143.444,Z 432.814,A -85,B 0,C 180,E1 -24586.545,E2 -24586.545} C_VEL
LIN {X 0,Y 143.272,Z 427.237,A -85,B 0,C 180,E1 -24591.89,E2 -24591.89} C_VEL
LIN {X 0,Y 146.051,Z 417.982,A -85,B 0,C 180,E1 -24600.617,E2 -24600.617} C_VEL
LIN {X 0,Y 146.588,Z 416.658,A -85,B 0,C 180,E1 -24601.828,E2 -24601.828} C_VEL
LIN {X 0,Y 146.487,Z 414.964,A -85,B 0,C 180,E1 -24603.371,E2 -24603.371} C_VEL
LIN {X 0,Y 144.791,Z 408.779,A -85,B 0,C 180,E1 -24609.124,E2 -24609.124} C_VEL
LIN {X 0,Y 143.348,Z 402.625,A -85,B 0,C 180,E1 -24615.189,E2 -24615.189} C_VEL
LIN {X 0,Y 143.114,Z 402.658,A -85,B 0,C 180,E1 -24621.787,E2 -24621.787} C_VEL
LIN {X 0,Y 143.106,Z 402.651,A -85,B 0,C 180,E1 -24625.44,E2 -24625.44} C_VEL
LIN {X 0,Y 142.465,Z 402.737,A -85,B 0,C 180,E1 -24627.788,E2 -24627.788} C_VEL
LIN {X 0,Y 140.86,Z 402.94,A -85,B 0,C 180,E1 -24630.102,E2 -24630.102} C_VEL
LIN {X 0,Y 137.127,Z 403.398,A -85,B 0,C 180,E1 -24634.829,E2 -24634.829} C_VEL
LIN {X 0,Y 136.202,Z 403.518,A -85,B 0,C 180,E1 -24637.323,E2 -24637.323} C_VEL
LIN {X 0,Y 136.19,Z 403.52,A -85,B 0,C 180,E1 -24638.168,E2 -24638.168} C_VEL
LIN {X 0,Y 136.252,Z 403.507,A -85,B 0,C 180,E1 -24641.972,E2 -24641.972} C_VEL
LIN {X 0,Y 136.501,Z 403.481,A -85,B 0,C 180,E1 -24648.115,E2 -24648.115} C_VEL
LIN {X 0,Y 136.609,Z 403.463,A -85,B 0,C 180,E1 -24651.122,E2 -24651.122} C_VEL
LIN {X 0,Y 137.135,Z 403.397,A -85,B 0,C 180,E1 -24660,E2 -24660} C_VEL
LIN {X 0,Y 136.609,Z 403.462,A -85,B 0,C 180,E1 -24668.879,E2 -24668.879} C_VEL
LIN {X 0,Y 136.493,Z 403.482,A -85,B 0,C 180,E1 -24671.959,E2 -24671.959} C_VEL
LIN {X 0,Y 136.257,Z 403.507,A -85,B 0,C 180,E1 -24678.028,E2 -24678.028} C_VEL
LIN {X 0,Y 136.199,Z 403.519,A -85,B 0,C 180,E1 -24681.75,E2 -24681.75} C_VEL
LIN {X 0,Y 136.119,Z 403.528,A -85,B 0,C 180,E1 -24688.631,E2 -24688.631} C_VEL
LIN {X 0,Y 136.045,Z 403.532,A -85,B 0,C 180,E1 -24694.629,E2 -24694.629} C_VEL
LIN {X 0,Y 136.033,Z 403.54,A -85,B 0,C 180,E1 -24699.2,E2 -24699.2} C_VEL
LIN {X 0,Y 135.997,Z 403.539,A -85,B 0,C 180,E1 -24703.658,E2 -24703.658} C_VEL
LIN {X 0,Y 136.032,Z 403.539,A -85,B 0,C 180,E1 -24707.807,E2 -24707.807} C_VEL
LIN {X 0,Y 136.056,Z 403.53,A -85,B 0,C 180,E1 -24711.695,E2 -24711.695} C_VEL
LIN {X 0,Y 136.091,Z 403.532,A -85,B 0,C 180,E1 -24715.718,E2 -24715.718} C_VEL
LIN {X 0,Y 136.148,Z 403.524,A -85,B 0,C 180,E1 -24722.317,E2 -24722.317} C_VEL
LIN {X 0,Y 136.279,Z 403.504,A -85,B 0,C 180,E1 -24728.839,E2 -24728.839} C_VEL
LIN {X 0,Y 136.294,Z 403.505,A -85,B 0,C 180,E1 -24735.059,E2 -24735.059} C_VEL
LIN {X 0,Y 136.498,Z 403.477,A -85,B 0,C 180,E1 -24738.115,E2 -24738.115} C_VEL
LIN {X 0,Y 136.594,Z 403.469,A -85,B 0,C 180,E1 -24741.121,E2 -24741.121} C_VEL
LIN {X 0,Y 137.137,Z 403.404,A -85,B 0,C 180,E1 -24750.001,E2 -24750.001} C_VEL
LIN {X 0,Y 136.554,Z 403.474,A -85,B 0,C 180,E1 -24758.883,E2 -24758.883} C_VEL
LIN {X 0,Y 136.442,Z 403.484,A -85,B 0,C 180,E1 -24761.891,E2 -24761.891} C_VEL
LIN {X 0,Y 136.249,Z 403.513,A -85,B 0,C 180,E1 -24768.029,E2 -24768.029} C_VEL
LIN {X 0,Y 136.201,Z 403.514,A -85,B 0,C 180,E1 -24771.75,E2 -24771.75} C_VEL
LIN {X 0,Y 136.103,Z 403.528,A -85,B 0,C 180,E1 -24778.617,E2 -24778.617} C_VEL
LIN {X 0,Y 136.081,Z 403.533,A -85,B 0,C 180,E1 -24784.619,E2 -24784.619} C_VEL
LIN {X 0,Y 136.053,Z 403.532,A -85,B 0,C 180,E1 -24789.209,E2 -24789.209} C_VEL
